    stNO_LENS[0].fEnergy := 5069.272832; stNO_LENS[0].fLow := 154.471527; stNO_LENS[0].fHigh := 156.009850; 
    stNO_LENS[1].fEnergy := 5079.421523; stNO_LENS[1].fLow := 153.906286; stNO_LENS[1].fHigh := 156.009850; 
    stNO_LENS[2].fEnergy := 5089.590532; stNO_LENS[2].fLow := 153.342381; stNO_LENS[2].fHigh := 156.009850; 
    stNO_LENS[3].fEnergy := 5099.779899; stNO_LENS[3].fLow := 152.779815; stNO_LENS[3].fHigh := 156.009850; 
    stNO_LENS[4].fEnergy := 5109.989665; stNO_LENS[4].fLow := 152.218592; stNO_LENS[4].fHigh := 156.009850; 
    stNO_LENS[5].fEnergy := 5120.219871; stNO_LENS[5].fLow := 151.658718; stNO_LENS[5].fHigh := 156.009850; 
    stNO_LENS[6].fEnergy := 5130.470558; stNO_LENS[6].fLow := 151.100196; stNO_LENS[6].fHigh := 156.009850; 
    stNO_LENS[7].fEnergy := 5140.741767; stNO_LENS[7].fLow := 150.543029; stNO_LENS[7].fHigh := 156.009850; 
    stNO_LENS[8].fEnergy := 5151.033539; stNO_LENS[8].fLow := 149.987222; stNO_LENS[8].fHigh := 156.009850; 
    stNO_LENS[9].fEnergy := 5161.345915; stNO_LENS[9].fLow := 149.432777; stNO_LENS[9].fHigh := 156.009850; 
    stNO_LENS[10].fEnergy := 5171.678936; stNO_LENS[10].fLow := 148.879700; stNO_LENS[10].fHigh := 156.009850; 
    stNO_LENS[11].fEnergy := 5182.032644; stNO_LENS[11].fLow := 148.327994; stNO_LENS[11].fHigh := 156.009850; 
    stNO_LENS[12].fEnergy := 5192.407080; stNO_LENS[12].fLow := 147.777661; stNO_LENS[12].fHigh := 156.009850; 
    stNO_LENS[13].fEnergy := 5202.802286; stNO_LENS[13].fLow := 147.228705; stNO_LENS[13].fHigh := 156.009850; 
    stNO_LENS[14].fEnergy := 5213.218304; stNO_LENS[14].fLow := 146.681131; stNO_LENS[14].fHigh := 156.009850; 
    stNO_LENS[15].fEnergy := 5223.655174; stNO_LENS[15].fLow := 146.134940; stNO_LENS[15].fHigh := 156.009850; 
    stNO_LENS[16].fEnergy := 5234.112938; stNO_LENS[16].fLow := 145.590136; stNO_LENS[16].fHigh := 156.022129; 
    stNO_LENS[17].fEnergy := 5244.591639; stNO_LENS[17].fLow := 145.046723; stNO_LENS[17].fHigh := 156.023236; 
    stNO_LENS[18].fEnergy := 5255.091319; stNO_LENS[18].fLow := 144.504703; stNO_LENS[18].fHigh := 156.013558; 
    stNO_LENS[19].fEnergy := 5265.612019; stNO_LENS[19].fLow := 143.964079; stNO_LENS[19].fHigh := 155.993480; 
    stNO_LENS[20].fEnergy := 5276.153781; stNO_LENS[20].fLow := 143.424854; stNO_LENS[20].fHigh := 155.963384; 
    stNO_LENS[21].fEnergy := 5286.716648; stNO_LENS[21].fLow := 142.887032; stNO_LENS[21].fHigh := 155.923643; 
    stNO_LENS[22].fEnergy := 5297.300661; stNO_LENS[22].fLow := 142.350614; stNO_LENS[22].fHigh := 155.874628; 
    stNO_LENS[23].fEnergy := 5307.905864; stNO_LENS[23].fLow := 141.815603; stNO_LENS[23].fHigh := 155.816705; 
    stNO_LENS[24].fEnergy := 5318.532299; stNO_LENS[24].fLow := 141.282002; stNO_LENS[24].fHigh := 155.750234; 
    stNO_LENS[25].fEnergy := 5329.180008; stNO_LENS[25].fLow := 140.749814; stNO_LENS[25].fHigh := 155.675570; 
    stNO_LENS[26].fEnergy := 5339.849033; stNO_LENS[26].fLow := 140.219040; stNO_LENS[26].fHigh := 155.593061; 
    stNO_LENS[27].fEnergy := 5350.539418; stNO_LENS[27].fLow := 139.689684; stNO_LENS[27].fHigh := 155.503052; 
    stNO_LENS[28].fEnergy := 5361.251205; stNO_LENS[28].fLow := 139.161747; stNO_LENS[28].fHigh := 155.405880; 
    stNO_LENS[29].fEnergy := 5371.984437; stNO_LENS[29].fLow := 138.635232; stNO_LENS[29].fHigh := 155.301878; 
    stNO_LENS[30].fEnergy := 5382.739157; stNO_LENS[30].fLow := 138.110142; stNO_LENS[30].fHigh := 155.191371; 
    stNO_LENS[31].fEnergy := 5393.515408; stNO_LENS[31].fLow := 137.586477; stNO_LENS[31].fHigh := 155.074681; 
    stNO_LENS[32].fEnergy := 5404.313233; stNO_LENS[32].fLow := 137.064240; stNO_LENS[32].fHigh := 154.952120; 
    stNO_LENS[33].fEnergy := 5415.132676; stNO_LENS[33].fLow := 136.543434; stNO_LENS[33].fHigh := 154.823998; 
    stNO_LENS[34].fEnergy := 5425.973779; stNO_LENS[34].fLow := 136.024059; stNO_LENS[34].fHigh := 154.690616; 
    stNO_LENS[35].fEnergy := 5436.836585; stNO_LENS[35].fLow := 135.506118; stNO_LENS[35].fHigh := 154.552270; 
    stNO_LENS[36].fEnergy := 5447.721139; stNO_LENS[36].fLow := 134.989613; stNO_LENS[36].fHigh := 154.409250; 
    stNO_LENS[37].fEnergy := 5458.627484; stNO_LENS[37].fLow := 134.474545; stNO_LENS[37].fHigh := 154.261839; 
    stNO_LENS[38].fEnergy := 5469.555664; stNO_LENS[38].fLow := 133.960916; stNO_LENS[38].fHigh := 154.110313; 
    stNO_LENS[39].fEnergy := 5480.505722; stNO_LENS[39].fLow := 133.448727; stNO_LENS[39].fHigh := 153.954945; 
    stNO_LENS[40].fEnergy := 5491.477701; stNO_LENS[40].fLow := 132.937980; stNO_LENS[40].fHigh := 153.795998; 
    stNO_LENS[41].fEnergy := 5502.471647; stNO_LENS[41].fLow := 132.428677; stNO_LENS[41].fHigh := 153.633731; 
    stNO_LENS[42].fEnergy := 5513.487603; stNO_LENS[42].fLow := 131.920818; stNO_LENS[42].fHigh := 153.468397; 
    stNO_LENS[43].fEnergy := 5524.525612; stNO_LENS[43].fLow := 131.414406; stNO_LENS[43].fHigh := 153.300240; 
    stNO_LENS[44].fEnergy := 5535.585720; stNO_LENS[44].fLow := 130.909441; stNO_LENS[44].fHigh := 153.129502; 
    stNO_LENS[45].fEnergy := 5546.667970; stNO_LENS[45].fLow := 130.405924; stNO_LENS[45].fHigh := 152.956416; 
    stNO_LENS[46].fEnergy := 5557.772406; stNO_LENS[46].fLow := 129.903857; stNO_LENS[46].fHigh := 152.781209; 
    stNO_LENS[47].fEnergy := 5568.899074; stNO_LENS[47].fLow := 129.403241; stNO_LENS[47].fHigh := 152.604103; 
    stNO_LENS[48].fEnergy := 5580.048018; stNO_LENS[48].fLow := 128.904077; stNO_LENS[48].fHigh := 152.425314; 
    stNO_LENS[49].fEnergy := 5591.219281; stNO_LENS[49].fLow := 128.406365; stNO_LENS[49].fHigh := 152.245051; 
    stNO_LENS[50].fEnergy := 5602.412910; stNO_LENS[50].fLow := 127.910107; stNO_LENS[50].fHigh := 152.063517; 
    stNO_LENS[51].fEnergy := 5613.628948; stNO_LENS[51].fLow := 127.415303; stNO_LENS[51].fHigh := 151.880912; 
    stNO_LENS[52].fEnergy := 5624.867440; stNO_LENS[52].fLow := 126.921955; stNO_LENS[52].fHigh := 151.697425; 
    stNO_LENS[53].fEnergy := 5636.128433; stNO_LENS[53].fLow := 126.430063; stNO_LENS[53].fHigh := 151.513245; 
    stNO_LENS[54].fEnergy := 5647.411969; stNO_LENS[54].fLow := 125.939627; stNO_LENS[54].fHigh := 151.328551; 
    stNO_LENS[55].fEnergy := 5658.718095; stNO_LENS[55].fLow := 125.450648; stNO_LENS[55].fHigh := 151.143518; 
    stNO_LENS[56].fEnergy := 5670.046857; stNO_LENS[56].fLow := 124.963127; stNO_LENS[56].fHigh := 150.958316; 
    stNO_LENS[57].fEnergy := 5681.398298; stNO_LENS[57].fLow := 124.477064; stNO_LENS[57].fHigh := 150.773109; 
    stNO_LENS[58].fEnergy := 5692.772465; stNO_LENS[58].fLow := 123.992460; stNO_LENS[58].fHigh := 150.588055; 
    stNO_LENS[59].fEnergy := 5704.169403; stNO_LENS[59].fLow := 123.509315; stNO_LENS[59].fHigh := 150.403307; 
    stNO_LENS[60].fEnergy := 5715.589158; stNO_LENS[60].fLow := 123.027630; stNO_LENS[60].fHigh := 150.219012; 
    stNO_LENS[61].fEnergy := 5727.031775; stNO_LENS[61].fLow := 122.547404; stNO_LENS[61].fHigh := 150.035315; 
    stNO_LENS[62].fEnergy := 5738.497300; stNO_LENS[62].fLow := 122.068638; stNO_LENS[62].fHigh := 149.852352; 
    stNO_LENS[63].fEnergy := 5749.985779; stNO_LENS[63].fLow := 121.591332; stNO_LENS[63].fHigh := 149.670256; 
    stNO_LENS[64].fEnergy := 5761.497259; stNO_LENS[64].fLow := 121.115486; stNO_LENS[64].fHigh := 149.489154; 
    stNO_LENS[65].fEnergy := 5773.031784; stNO_LENS[65].fLow := 120.641101; stNO_LENS[65].fHigh := 149.309169; 
    stNO_LENS[66].fEnergy := 5784.589401; stNO_LENS[66].fLow := 120.168176; stNO_LENS[66].fHigh := 149.130419; 
    stNO_LENS[67].fEnergy := 5796.170157; stNO_LENS[67].fLow := 119.696711; stNO_LENS[67].fHigh := 148.953017; 
    stNO_LENS[68].fEnergy := 5807.774097; stNO_LENS[68].fLow := 119.226706; stNO_LENS[68].fHigh := 148.777072; 
    stNO_LENS[69].fEnergy := 5819.401269; stNO_LENS[69].fLow := 118.758161; stNO_LENS[69].fHigh := 148.602686; 
    stNO_LENS[70].fEnergy := 5831.051718; stNO_LENS[70].fLow := 118.291076; stNO_LENS[70].fHigh := 148.429960; 
    stNO_LENS[71].fEnergy := 5842.725491; stNO_LENS[71].fLow := 117.825451; stNO_LENS[71].fHigh := 148.258988; 
    stNO_LENS[72].fEnergy := 5854.422635; stNO_LENS[72].fLow := 117.361285; stNO_LENS[72].fHigh := 148.089861; 
    stNO_LENS[73].fEnergy := 5866.143197; stNO_LENS[73].fLow := 116.898578; stNO_LENS[73].fHigh := 147.922666; 
    stNO_LENS[74].fEnergy := 5877.887224; stNO_LENS[74].fLow := 116.437330; stNO_LENS[74].fHigh := 147.757483; 
    stNO_LENS[75].fEnergy := 5889.654762; stNO_LENS[75].fLow := 115.977540; stNO_LENS[75].fHigh := 147.594392; 
    stNO_LENS[76].fEnergy := 5901.445859; stNO_LENS[76].fLow := 115.519207; stNO_LENS[76].fHigh := 147.433465; 
    stNO_LENS[77].fEnergy := 5913.260561; stNO_LENS[77].fLow := 115.062332; stNO_LENS[77].fHigh := 147.274774; 
    stNO_LENS[78].fEnergy := 5925.098917; stNO_LENS[78].fLow := 114.606914; stNO_LENS[78].fHigh := 147.118383; 
    stNO_LENS[79].fEnergy := 5936.960973; stNO_LENS[79].fLow := 114.152952; stNO_LENS[79].fHigh := 146.964356; 
    stNO_LENS[80].fEnergy := 5948.846776; stNO_LENS[80].fLow := 113.700445; stNO_LENS[80].fHigh := 146.812749; 
    stNO_LENS[81].fEnergy := 5960.756375; stNO_LENS[81].fLow := 113.249392; stNO_LENS[81].fHigh := 146.663619; 
    stNO_LENS[82].fEnergy := 5972.689818; stNO_LENS[82].fLow := 112.799794; stNO_LENS[82].fHigh := 146.517015; 
    stNO_LENS[83].fEnergy := 5984.647151; stNO_LENS[83].fLow := 112.351649; stNO_LENS[83].fHigh := 146.372987; 
    stNO_LENS[84].fEnergy := 5996.628422; stNO_LENS[84].fLow := 111.904956; stNO_LENS[84].fHigh := 146.231576; 
    stNO_LENS[85].fEnergy := 6008.633680; stNO_LENS[85].fLow := 111.459715; stNO_LENS[85].fHigh := 146.092825; 
    stNO_LENS[86].fEnergy := 6020.662973; stNO_LENS[86].fLow := 111.015925; stNO_LENS[86].fHigh := 145.956770; 
    stNO_LENS[87].fEnergy := 6032.716348; stNO_LENS[87].fLow := 110.573584; stNO_LENS[87].fHigh := 145.823445; 
    stNO_LENS[88].fEnergy := 6044.793854; stNO_LENS[88].fLow := 110.132692; stNO_LENS[88].fHigh := 145.692881; 
    stNO_LENS[89].fEnergy := 6056.895540; stNO_LENS[89].fLow := 109.693247; stNO_LENS[89].fHigh := 145.565105; 
    stNO_LENS[90].fEnergy := 6069.021453; stNO_LENS[90].fLow := 109.255249; stNO_LENS[90].fHigh := 145.440142; 
    stNO_LENS[91].fEnergy := 6081.171642; stNO_LENS[91].fLow := 108.818697; stNO_LENS[91].fHigh := 145.318013; 
    stNO_LENS[92].fEnergy := 6093.346156; stNO_LENS[92].fLow := 108.383589; stNO_LENS[92].fHigh := 145.198736; 
    stNO_LENS[93].fEnergy := 6105.545043; stNO_LENS[93].fLow := 107.949924; stNO_LENS[93].fHigh := 145.082327; 
    stNO_LENS[94].fEnergy := 6117.768352; stNO_LENS[94].fLow := 107.517701; stNO_LENS[94].fHigh := 144.968799; 
    stNO_LENS[95].fEnergy := 6130.016132; stNO_LENS[95].fLow := 107.086918; stNO_LENS[95].fHigh := 144.858160; 
    stNO_LENS[96].fEnergy := 6142.288433; stNO_LENS[96].fLow := 106.657575; stNO_LENS[96].fHigh := 144.750419; 
    stNO_LENS[97].fEnergy := 6154.585303; stNO_LENS[97].fLow := 106.229670; stNO_LENS[97].fHigh := 144.645579; 
    stNO_LENS[98].fEnergy := 6166.906791; stNO_LENS[98].fLow := 105.803201; stNO_LENS[98].fHigh := 144.543642; 
    stNO_LENS[99].fEnergy := 6179.252946; stNO_LENS[99].fLow := 105.378168; stNO_LENS[99].fHigh := 144.444606; 
    stNO_LENS[100].fEnergy := 6191.623819; stNO_LENS[100].fLow := 104.954569; stNO_LENS[100].fHigh := 144.348469; 
    stNO_LENS[101].fEnergy := 6204.019458; stNO_LENS[101].fLow := 104.532401; stNO_LENS[101].fHigh := 144.255225; 
    stNO_LENS[102].fEnergy := 6216.439913; stNO_LENS[102].fLow := 104.111665; stNO_LENS[102].fHigh := 144.164864; 
    stNO_LENS[103].fEnergy := 6228.885234; stNO_LENS[103].fLow := 103.692358; stNO_LENS[103].fHigh := 144.077376; 
    stNO_LENS[104].fEnergy := 6241.355471; stNO_LENS[104].fLow := 103.274478; stNO_LENS[104].fHigh := 143.992747; 
    stNO_LENS[105].fEnergy := 6253.850673; stNO_LENS[105].fLow := 102.858024; stNO_LENS[105].fHigh := 143.910962; 
    stNO_LENS[106].fEnergy := 6266.370890; stNO_LENS[106].fLow := 102.442995; stNO_LENS[106].fHigh := 143.832003; 
    stNO_LENS[107].fEnergy := 6278.916173; stNO_LENS[107].fLow := 102.029389; stNO_LENS[107].fHigh := 143.755850; 
    stNO_LENS[108].fEnergy := 6291.486572; stNO_LENS[108].fLow := 101.617203; stNO_LENS[108].fHigh := 143.682481; 
    stNO_LENS[109].fEnergy := 6304.082136; stNO_LENS[109].fLow := 101.206436; stNO_LENS[109].fHigh := 143.611870; 
    stNO_LENS[110].fEnergy := 6316.702917; stNO_LENS[110].fLow := 100.797087; stNO_LENS[110].fHigh := 143.543993; 
    stNO_LENS[111].fEnergy := 6329.348965; stNO_LENS[111].fLow := 100.389154; stNO_LENS[111].fHigh := 143.478819; 
    stNO_LENS[112].fEnergy := 6342.020330; stNO_LENS[112].fLow := 99.982634; stNO_LENS[112].fHigh := 143.416319; 
    stNO_LENS[113].fEnergy := 6354.717063; stNO_LENS[113].fLow := 99.577526; stNO_LENS[113].fHigh := 143.356460; 
    stNO_LENS[114].fEnergy := 6367.439215; stNO_LENS[114].fLow := 99.173828; stNO_LENS[114].fHigh := 143.299207; 
    stNO_LENS[115].fEnergy := 6380.186837; stNO_LENS[115].fLow := 98.771538; stNO_LENS[115].fHigh := 143.244524; 
    stNO_LENS[116].fEnergy := 6392.959979; stNO_LENS[116].fLow := 98.370654; stNO_LENS[116].fHigh := 143.192372; 
    stNO_LENS[117].fEnergy := 6405.758694; stNO_LENS[117].fLow := 97.971174; stNO_LENS[117].fHigh := 143.142713; 
    stNO_LENS[118].fEnergy := 6418.583031; stNO_LENS[118].fLow := 97.573096; stNO_LENS[118].fHigh := 143.095503; 
    stNO_LENS[119].fEnergy := 6431.433043; stNO_LENS[119].fLow := 97.176418; stNO_LENS[119].fHigh := 143.050699; 
    stNO_LENS[120].fEnergy := 6444.308780; stNO_LENS[120].fLow := 96.781138; stNO_LENS[120].fHigh := 143.008256; 
    stNO_LENS[121].fEnergy := 6457.210295; stNO_LENS[121].fLow := 96.387254; stNO_LENS[121].fHigh := 142.968127; 
    stNO_LENS[122].fEnergy := 6470.137639; stNO_LENS[122].fLow := 95.994763; stNO_LENS[122].fHigh := 142.930263; 
    stNO_LENS[123].fEnergy := 6483.090863; stNO_LENS[123].fLow := 95.603664; stNO_LENS[123].fHigh := 142.894614; 
    stNO_LENS[124].fEnergy := 6496.070019; stNO_LENS[124].fLow := 95.213954; stNO_LENS[124].fHigh := 142.861129; 
    stNO_LENS[125].fEnergy := 6509.075160; stNO_LENS[125].fLow := 94.825631; stNO_LENS[125].fHigh := 142.829753; 
    stNO_LENS[126].fEnergy := 6522.106337; stNO_LENS[126].fLow := 94.438693; stNO_LENS[126].fHigh := 142.800431; 
    stNO_LENS[127].fEnergy := 6535.163603; stNO_LENS[127].fLow := 94.053137; stNO_LENS[127].fHigh := 142.773109; 
    stNO_LENS[128].fEnergy := 6548.247009; stNO_LENS[128].fLow := 93.668962; stNO_LENS[128].fHigh := 142.747727; 
    stNO_LENS[129].fEnergy := 6561.356609; stNO_LENS[129].fLow := 93.286164; stNO_LENS[129].fHigh := 142.724228; 
    stNO_LENS[130].fEnergy := 6574.492453; stNO_LENS[130].fLow := 92.904742; stNO_LENS[130].fHigh := 142.702549; 
    stNO_LENS[131].fEnergy := 6587.654596; stNO_LENS[131].fLow := 92.524694; stNO_LENS[131].fHigh := 142.682630; 
    stNO_LENS[132].fEnergy := 6600.843089; stNO_LENS[132].fLow := 92.146016; stNO_LENS[132].fHigh := 142.664407; 
    stNO_LENS[133].fEnergy := 6614.057986; stNO_LENS[133].fLow := 91.768706; stNO_LENS[133].fHigh := 142.647816; 
    stNO_LENS[134].fEnergy := 6627.299339; stNO_LENS[134].fLow := 91.392763; stNO_LENS[134].fHigh := 142.632791; 
    stNO_LENS[135].fEnergy := 6640.567201; stNO_LENS[135].fLow := 91.018183; stNO_LENS[135].fHigh := 142.619266; 
    stNO_LENS[136].fEnergy := 6653.861625; stNO_LENS[136].fLow := 90.644964; stNO_LENS[136].fHigh := 142.607171; 
    stNO_LENS[137].fEnergy := 6667.182665; stNO_LENS[137].fLow := 90.273103; stNO_LENS[137].fHigh := 142.596440; 
    stNO_LENS[138].fEnergy := 6680.530374; stNO_LENS[138].fLow := 89.902598; stNO_LENS[138].fHigh := 142.587000; 
    stNO_LENS[139].fEnergy := 6693.904804; stNO_LENS[139].fLow := 89.533447; stNO_LENS[139].fHigh := 142.578781; 
    stNO_LENS[140].fEnergy := 6707.306011; stNO_LENS[140].fLow := 89.165646; stNO_LENS[140].fHigh := 142.571711; 
    stNO_LENS[141].fEnergy := 6720.734046; stNO_LENS[141].fLow := 88.799194; stNO_LENS[141].fHigh := 142.565716; 
    stNO_LENS[142].fEnergy := 6734.188965; stNO_LENS[142].fLow := 88.434088; stNO_LENS[142].fHigh := 142.560721; 
    stNO_LENS[143].fEnergy := 6747.670820; stNO_LENS[143].fLow := 88.070324; stNO_LENS[143].fHigh := 142.556653; 
    stNO_LENS[144].fEnergy := 6761.179666; stNO_LENS[144].fLow := 87.707901; stNO_LENS[144].fHigh := 142.553434; 
    stNO_LENS[145].fEnergy := 6774.715557; stNO_LENS[145].fLow := 87.346815; stNO_LENS[145].fHigh := 142.550988; 
    stNO_LENS[146].fEnergy := 6788.278546; stNO_LENS[146].fLow := 86.987064; stNO_LENS[146].fHigh := 142.549237; 
    stNO_LENS[147].fEnergy := 6801.868689; stNO_LENS[147].fLow := 86.628646; stNO_LENS[147].fHigh := 142.548102; 
    stNO_LENS[148].fEnergy := 6815.486039; stNO_LENS[148].fLow := 86.271557; stNO_LENS[148].fHigh := 142.547505; 
    stNO_LENS[149].fEnergy := 6829.130652; stNO_LENS[149].fLow := 85.915795; stNO_LENS[149].fHigh := 142.547365; 
    stNO_LENS[150].fEnergy := 6842.802580; stNO_LENS[150].fLow := 85.561357; stNO_LENS[150].fHigh := 142.547602; 
    stNO_LENS[151].fEnergy := 6856.501880; stNO_LENS[151].fLow := 85.208240; stNO_LENS[151].fHigh := 142.548134; 
    stNO_LENS[152].fEnergy := 6870.228606; stNO_LENS[152].fLow := 84.856441; stNO_LENS[152].fHigh := 142.548880; 
    stNO_LENS[153].fEnergy := 6883.982813; stNO_LENS[153].fLow := 84.505959; stNO_LENS[153].fHigh := 142.549757; 
    stNO_LENS[154].fEnergy := 6897.764556; stNO_LENS[154].fLow := 84.156788; stNO_LENS[154].fHigh := 142.550682; 
    stNO_LENS[155].fEnergy := 6911.573889; stNO_LENS[155].fLow := 83.808928; stNO_LENS[155].fHigh := 142.551572; 
    stNO_LENS[156].fEnergy := 6925.410870; stNO_LENS[156].fLow := 83.462375; stNO_LENS[156].fHigh := 142.552342; 
    stNO_LENS[157].fEnergy := 6939.275551; stNO_LENS[157].fLow := 83.117126; stNO_LENS[157].fHigh := 142.552910; 
    stNO_LENS[158].fEnergy := 6953.167990; stNO_LENS[158].fLow := 82.773178; stNO_LENS[158].fHigh := 142.553189; 
    stNO_LENS[159].fEnergy := 6967.088242; stNO_LENS[159].fLow := 82.430528; stNO_LENS[159].fHigh := 142.553096; 
    stNO_LENS[160].fEnergy := 6981.036362; stNO_LENS[160].fLow := 82.089174; stNO_LENS[160].fHigh := 142.552545; 
    stNO_LENS[161].fEnergy := 6995.012406; stNO_LENS[161].fLow := 81.749112; stNO_LENS[161].fHigh := 142.551451; 
    stNO_LENS[162].fEnergy := 7009.016430; stNO_LENS[162].fLow := 81.410340; stNO_LENS[162].fHigh := 142.549728; 
    stNO_LENS[163].fEnergy := 7023.048490; stNO_LENS[163].fLow := 81.072854; stNO_LENS[163].fHigh := 142.547290; 
    stNO_LENS[164].fEnergy := 7037.108643; stNO_LENS[164].fLow := 80.736651; stNO_LENS[164].fHigh := 142.544051; 
    stNO_LENS[165].fEnergy := 7051.196944; stNO_LENS[165].fLow := 80.401730; stNO_LENS[165].fHigh := 142.539926; 
    stNO_LENS[166].fEnergy := 7065.313449; stNO_LENS[166].fLow := 80.068085; stNO_LENS[166].fHigh := 142.534829; 
    stNO_LENS[167].fEnergy := 7079.458216; stNO_LENS[167].fLow := 79.735715; stNO_LENS[167].fHigh := 142.528674; 
    stNO_LENS[168].fEnergy := 7093.631301; stNO_LENS[168].fLow := 79.404617; stNO_LENS[168].fHigh := 142.521375; 
    stNO_LENS[169].fEnergy := 7107.832760; stNO_LENS[169].fLow := 79.074786; stNO_LENS[169].fHigh := 142.512847; 
    stNO_LENS[170].fEnergy := 7122.062651; stNO_LENS[170].fLow := 78.746221; stNO_LENS[170].fHigh := 142.503004; 
    stNO_LENS[171].fEnergy := 7136.321030; stNO_LENS[171].fLow := 78.418918; stNO_LENS[171].fHigh := 142.491760; 
    stNO_LENS[172].fEnergy := 7150.607954; stNO_LENS[172].fLow := 78.092875; stNO_LENS[172].fHigh := 142.479032; 
    stNO_LENS[173].fEnergy := 7164.923481; stNO_LENS[173].fLow := 77.768087; stNO_LENS[173].fHigh := 142.464734; 
    stNO_LENS[174].fEnergy := 7179.267667; stNO_LENS[174].fLow := 77.444552; stNO_LENS[174].fHigh := 142.448782; 
    stNO_LENS[175].fEnergy := 7193.640571; stNO_LENS[175].fLow := 77.122267; stNO_LENS[175].fHigh := 142.431092; 
    stNO_LENS[176].fEnergy := 7208.042249; stNO_LENS[176].fLow := 76.801228; stNO_LENS[176].fHigh := 142.411581; 
    stNO_LENS[177].fEnergy := 7222.472759; stNO_LENS[177].fLow := 76.481433; stNO_LENS[177].fHigh := 142.390166; 
    stNO_LENS[178].fEnergy := 7236.932159; stNO_LENS[178].fLow := 76.162878; stNO_LENS[178].fHigh := 142.366765; 
    stNO_LENS[179].fEnergy := 7251.420507; stNO_LENS[179].fLow := 75.845560; stNO_LENS[179].fHigh := 142.341297; 
    stNO_LENS[180].fEnergy := 7265.937860; stNO_LENS[180].fLow := 75.529476; stNO_LENS[180].fHigh := 142.313679; 
    stNO_LENS[181].fEnergy := 7280.484278; stNO_LENS[181].fLow := 75.214623; stNO_LENS[181].fHigh := 142.283833; 
    stNO_LENS[182].fEnergy := 7295.059817; stNO_LENS[182].fLow := 74.900997; stNO_LENS[182].fHigh := 142.251678; 
    stNO_LENS[183].fEnergy := 7309.664536; stNO_LENS[183].fLow := 74.588595; stNO_LENS[183].fHigh := 142.217136; 
    stNO_LENS[184].fEnergy := 7324.298495; stNO_LENS[184].fLow := 74.277415; stNO_LENS[184].fHigh := 142.180129; 
    stNO_LENS[185].fEnergy := 7338.961750; stNO_LENS[185].fLow := 73.967452; stNO_LENS[185].fHigh := 142.140581; 
    stNO_LENS[186].fEnergy := 7353.654361; stNO_LENS[186].fLow := 73.658704; stNO_LENS[186].fHigh := 142.098415; 
    stNO_LENS[187].fEnergy := 7368.376387; stNO_LENS[187].fLow := 73.351168; stNO_LENS[187].fHigh := 142.053558; 
    stNO_LENS[188].fEnergy := 7383.127886; stNO_LENS[188].fLow := 73.044839; stNO_LENS[188].fHigh := 142.005934; 
    stNO_LENS[189].fEnergy := 7397.908918; stNO_LENS[189].fLow := 72.739716; stNO_LENS[189].fHigh := 141.955472; 
    stNO_LENS[190].fEnergy := 7412.719542; stNO_LENS[190].fLow := 72.435793; stNO_LENS[190].fHigh := 141.902101; 
    stNO_LENS[191].fEnergy := 7427.559816; stNO_LENS[191].fLow := 72.133070; stNO_LENS[191].fHigh := 141.845750; 
    stNO_LENS[192].fEnergy := 7442.429801; stNO_LENS[192].fLow := 71.831541; stNO_LENS[192].fHigh := 141.786350; 
    stNO_LENS[193].fEnergy := 7457.329555; stNO_LENS[193].fLow := 71.531203; stNO_LENS[193].fHigh := 141.723834; 
    stNO_LENS[194].fEnergy := 7472.259139; stNO_LENS[194].fLow := 71.232055; stNO_LENS[194].fHigh := 141.658137; 
    stNO_LENS[195].fEnergy := 7487.218612; stNO_LENS[195].fLow := 70.934091; stNO_LENS[195].fHigh := 141.589194; 
    stNO_LENS[196].fEnergy := 7502.208033; stNO_LENS[196].fLow := 70.637309; stNO_LENS[196].fHigh := 141.516941; 
    stNO_LENS[197].fEnergy := 7517.227464; stNO_LENS[197].fLow := 70.341705; stNO_LENS[197].fHigh := 141.441317; 
    stNO_LENS[198].fEnergy := 7532.276963; stNO_LENS[198].fLow := 70.047277; stNO_LENS[198].fHigh := 141.362263; 
    stNO_LENS[199].fEnergy := 7547.356592; stNO_LENS[199].fLow := 69.754020; stNO_LENS[199].fHigh := 141.279720; 
    stNO_LENS[200].fEnergy := 7562.466410; stNO_LENS[200].fLow := 69.461932; stNO_LENS[200].fHigh := 141.193632; 
    stNO_LENS[201].fEnergy := 7577.606478; stNO_LENS[201].fLow := 69.171009; stNO_LENS[201].fHigh := 141.103944; 
    stNO_LENS[202].fEnergy := 7592.776856; stNO_LENS[202].fLow := 68.881248; stNO_LENS[202].fHigh := 141.010603; 
    stNO_LENS[203].fEnergy := 7607.977605; stNO_LENS[203].fLow := 68.592645; stNO_LENS[203].fHigh := 140.913560; 
    stNO_LENS[204].fEnergy := 7623.208787; stNO_LENS[204].fLow := 68.305197; stNO_LENS[204].fHigh := 140.812763; 
    stNO_LENS[205].fEnergy := 7638.470461; stNO_LENS[205].fLow := 68.018901; stNO_LENS[205].fHigh := 140.708168; 
    stNO_LENS[206].fEnergy := 7653.762689; stNO_LENS[206].fLow := 67.733753; stNO_LENS[206].fHigh := 140.599727; 
    stNO_LENS[207].fEnergy := 7669.085532; stNO_LENS[207].fLow := 67.449750; stNO_LENS[207].fHigh := 140.487400; 
    stNO_LENS[208].fEnergy := 7684.439051; stNO_LENS[208].fLow := 67.166889; stNO_LENS[208].fHigh := 140.371143; 
    stNO_LENS[209].fEnergy := 7699.823309; stNO_LENS[209].fLow := 66.885165; stNO_LENS[209].fHigh := 140.250920; 
    stNO_LENS[210].fEnergy := 7715.238365; stNO_LENS[210].fLow := 66.604577; stNO_LENS[210].fHigh := 140.126694; 
    stNO_LENS[211].fEnergy := 7730.684283; stNO_LENS[211].fLow := 66.325120; stNO_LENS[211].fHigh := 139.998430; 
    stNO_LENS[212].fEnergy := 7746.161123; stNO_LENS[212].fLow := 66.046791; stNO_LENS[212].fHigh := 139.866096; 
    stNO_LENS[213].fEnergy := 7761.668948; stNO_LENS[213].fLow := 65.769586; stNO_LENS[213].fHigh := 139.729663; 
    stNO_LENS[214].fEnergy := 7777.207819; stNO_LENS[214].fLow := 65.493503; stNO_LENS[214].fHigh := 139.589104; 
    stNO_LENS[215].fEnergy := 7792.777800; stNO_LENS[215].fLow := 65.218537; stNO_LENS[215].fHigh := 139.444394; 
    stNO_LENS[216].fEnergy := 7808.378951; stNO_LENS[216].fLow := 64.944686; stNO_LENS[216].fHigh := 139.295510; 
    stNO_LENS[217].fEnergy := 7824.011336; stNO_LENS[217].fLow := 64.671946; stNO_LENS[217].fHigh := 139.142433; 
    stNO_LENS[218].fEnergy := 7839.675018; stNO_LENS[218].fLow := 64.400313; stNO_LENS[218].fHigh := 138.985145; 
    stNO_LENS[219].fEnergy := 7855.370057; stNO_LENS[219].fLow := 64.129785; stNO_LENS[219].fHigh := 138.823631; 
    stNO_LENS[220].fEnergy := 7871.096519; stNO_LENS[220].fLow := 63.860357; stNO_LENS[220].fHigh := 138.657880; 
    stNO_LENS[221].fEnergy := 7886.854464; stNO_LENS[221].fLow := 63.592027; stNO_LENS[221].fHigh := 138.487882; 
    stNO_LENS[222].fEnergy := 7902.643958; stNO_LENS[222].fLow := 63.324790; stNO_LENS[222].fHigh := 138.313630; 
    stNO_LENS[223].fEnergy := 7918.465061; stNO_LENS[223].fLow := 63.058644; stNO_LENS[223].fHigh := 138.135119; 
    stNO_LENS[224].fEnergy := 7934.317839; stNO_LENS[224].fLow := 62.793585; stNO_LENS[224].fHigh := 137.952349; 
    stNO_LENS[225].fEnergy := 7950.202354; stNO_LENS[225].fLow := 62.529610; stNO_LENS[225].fHigh := 137.765320; 
    stNO_LENS[226].fEnergy := 7966.118670; stNO_LENS[226].fLow := 62.266715; stNO_LENS[226].fHigh := 137.608060; 
    stNO_LENS[227].fEnergy := 7982.066850; stNO_LENS[227].fLow := 62.004896; stNO_LENS[227].fHigh := 137.048845; 
    stNO_LENS[228].fEnergy := 7998.046958; stNO_LENS[228].fLow := 61.744151; stNO_LENS[228].fHigh := 136.491790; 
    stNO_LENS[229].fEnergy := 8014.059059; stNO_LENS[229].fLow := 61.484476; stNO_LENS[229].fHigh := 135.936902; 
    stNO_LENS[230].fEnergy := 8030.103216; stNO_LENS[230].fLow := 61.225868; stNO_LENS[230].fHigh := 135.384186; 
    stNO_LENS[231].fEnergy := 8046.179493; stNO_LENS[231].fLow := 60.968322; stNO_LENS[231].fHigh := 134.833648; 
    stNO_LENS[232].fEnergy := 8062.287955; stNO_LENS[232].fLow := 60.711836; stNO_LENS[232].fHigh := 134.285293; 
    stNO_LENS[233].fEnergy := 8078.428667; stNO_LENS[233].fLow := 60.456407; stNO_LENS[233].fHigh := 133.739125; 
    stNO_LENS[234].fEnergy := 8094.601692; stNO_LENS[234].fLow := 60.202030; stNO_LENS[234].fHigh := 133.195147; 
    stNO_LENS[235].fEnergy := 8110.807095; stNO_LENS[235].fLow := 59.948702; stNO_LENS[235].fHigh := 132.653363; 
    stNO_LENS[236].fEnergy := 8127.044942; stNO_LENS[236].fLow := 59.696420; stNO_LENS[236].fHigh := 132.113775; 
    stNO_LENS[237].fEnergy := 8143.315296; stNO_LENS[237].fLow := 59.445181; stNO_LENS[237].fHigh := 131.576385; 
    stNO_LENS[238].fEnergy := 8159.618224; stNO_LENS[238].fLow := 59.194981; stNO_LENS[238].fHigh := 131.041195; 
    stNO_LENS[239].fEnergy := 8175.953791; stNO_LENS[239].fLow := 58.945817; stNO_LENS[239].fHigh := 130.508206; 
    stNO_LENS[240].fEnergy := 8192.322061; stNO_LENS[240].fLow := 58.697684; stNO_LENS[240].fHigh := 129.977418; 
    stNO_LENS[241].fEnergy := 8208.723101; stNO_LENS[241].fLow := 58.450581; stNO_LENS[241].fHigh := 129.448832; 
    stNO_LENS[242].fEnergy := 8225.156976; stNO_LENS[242].fLow := 58.204503; stNO_LENS[242].fHigh := 128.922447; 
    stNO_LENS[243].fEnergy := 8241.623751; stNO_LENS[243].fLow := 57.959446; stNO_LENS[243].fHigh := 128.398263; 
    stNO_LENS[244].fEnergy := 8258.123493; stNO_LENS[244].fLow := 57.715408; stNO_LENS[244].fHigh := 127.876278; 
    stNO_LENS[245].fEnergy := 8274.656267; stNO_LENS[245].fLow := 57.472386; stNO_LENS[245].fHigh := 127.356491; 
    stNO_LENS[246].fEnergy := 8291.222140; stNO_LENS[246].fLow := 57.230375; stNO_LENS[246].fHigh := 126.838900; 
    stNO_LENS[247].fEnergy := 8307.821178; stNO_LENS[247].fLow := 56.989372; stNO_LENS[247].fHigh := 126.323503; 
    stNO_LENS[248].fEnergy := 8324.453447; stNO_LENS[248].fLow := 56.749374; stNO_LENS[248].fHigh := 125.810298; 
    stNO_LENS[249].fEnergy := 8341.119014; stNO_LENS[249].fLow := 56.510377; stNO_LENS[249].fHigh := 125.299281; 
    stNO_LENS[250].fEnergy := 8357.817945; stNO_LENS[250].fLow := 56.272379; stNO_LENS[250].fHigh := 124.790450; 
    stNO_LENS[251].fEnergy := 8374.550308; stNO_LENS[251].fLow := 56.035375; stNO_LENS[251].fHigh := 124.283800; 
    stNO_LENS[252].fEnergy := 8391.316169; stNO_LENS[252].fLow := 55.799362; stNO_LENS[252].fHigh := 123.779328; 
    stNO_LENS[253].fEnergy := 8408.115595; stNO_LENS[253].fLow := 55.564337; stNO_LENS[253].fHigh := 123.277031; 
    stNO_LENS[254].fEnergy := 8424.948653; stNO_LENS[254].fLow := 55.330296; stNO_LENS[254].fHigh := 122.776902; 
    stNO_LENS[255].fEnergy := 8441.815412; stNO_LENS[255].fLow := 55.097236; stNO_LENS[255].fHigh := 122.278938; 
    stNO_LENS[256].fEnergy := 8458.715938; stNO_LENS[256].fLow := 54.865154; stNO_LENS[256].fHigh := 121.783134; 
    stNO_LENS[257].fEnergy := 8475.650298; stNO_LENS[257].fLow := 54.634046; stNO_LENS[257].fHigh := 121.289485; 
    stNO_LENS[258].fEnergy := 8492.618561; stNO_LENS[258].fLow := 54.403909; stNO_LENS[258].fHigh := 120.797985; 
    stNO_LENS[259].fEnergy := 8509.620795; stNO_LENS[259].fLow := 54.174739; stNO_LENS[259].fHigh := 120.308629; 
    stNO_LENS[260].fEnergy := 8526.657067; stNO_LENS[260].fLow := 53.946533; stNO_LENS[260].fHigh := 119.821410; 
    stNO_LENS[261].fEnergy := 8543.727446; stNO_LENS[261].fLow := 53.719288; stNO_LENS[261].fHigh := 119.336324; 
    stNO_LENS[262].fEnergy := 8560.832000; stNO_LENS[262].fLow := 53.493000; stNO_LENS[262].fHigh := 118.853363; 
    stNO_LENS[263].fEnergy := 8577.970797; stNO_LENS[263].fLow := 53.267666; stNO_LENS[263].fHigh := 118.372521; 
    stNO_LENS[264].fEnergy := 8595.143906; stNO_LENS[264].fLow := 53.043282; stNO_LENS[264].fHigh := 117.893792; 
    stNO_LENS[265].fEnergy := 8612.351395; stNO_LENS[265].fLow := 52.819845; stNO_LENS[265].fHigh := 117.417168; 
    stNO_LENS[266].fEnergy := 8629.593334; stNO_LENS[266].fLow := 52.597352; stNO_LENS[266].fHigh := 116.942644; 
    stNO_LENS[267].fEnergy := 8646.869792; stNO_LENS[267].fLow := 52.375800; stNO_LENS[267].fHigh := 116.470212; 
    stNO_LENS[268].fEnergy := 8664.180837; stNO_LENS[268].fLow := 52.155184; stNO_LENS[268].fHigh := 115.999864; 
    stNO_LENS[269].fEnergy := 8681.526538; stNO_LENS[269].fLow := 51.935503; stNO_LENS[269].fHigh := 115.531593; 
    stNO_LENS[270].fEnergy := 8698.906966; stNO_LENS[270].fLow := 51.716751; stNO_LENS[270].fHigh := 115.065393; 
    stNO_LENS[271].fEnergy := 8716.322189; stNO_LENS[271].fLow := 51.498926; stNO_LENS[271].fHigh := 114.601255; 
    stNO_LENS[272].fEnergy := 8733.772278; stNO_LENS[272].fLow := 51.282026; stNO_LENS[272].fHigh := 114.139171; 
    stNO_LENS[273].fEnergy := 8751.257302; stNO_LENS[273].fLow := 51.066045; stNO_LENS[273].fHigh := 113.679134; 
    stNO_LENS[274].fEnergy := 8768.777330; stNO_LENS[274].fLow := 50.850981; stNO_LENS[274].fHigh := 113.221136; 
    stNO_LENS[275].fEnergy := 8786.332434; stNO_LENS[275].fLow := 50.636831; stNO_LENS[275].fHigh := 112.765169; 
    stNO_LENS[276].fEnergy := 8803.922684; stNO_LENS[276].fLow := 50.423591; stNO_LENS[276].fHigh := 112.311224; 
    stNO_LENS[277].fEnergy := 8821.548149; stNO_LENS[277].fLow := 50.211258; stNO_LENS[277].fHigh := 111.859294; 
    stNO_LENS[278].fEnergy := 8839.208900; stNO_LENS[278].fLow := 49.999829; stNO_LENS[278].fHigh := 111.409371; 
    stNO_LENS[279].fEnergy := 8856.905008; stNO_LENS[279].fLow := 49.789301; stNO_LENS[279].fHigh := 110.961445; 
    stNO_LENS[280].fEnergy := 8874.636543; stNO_LENS[280].fLow := 49.579669; stNO_LENS[280].fHigh := 110.515509; 
    stNO_LENS[281].fEnergy := 8892.403578; stNO_LENS[281].fLow := 49.370931; stNO_LENS[281].fHigh := 110.071554; 
    stNO_LENS[282].fEnergy := 8910.206181; stNO_LENS[282].fLow := 49.163083; stNO_LENS[282].fHigh := 109.629572; 
    stNO_LENS[283].fEnergy := 8928.044426; stNO_LENS[283].fLow := 48.956123; stNO_LENS[283].fHigh := 109.189554; 
    stNO_LENS[284].fEnergy := 8945.918383; stNO_LENS[284].fLow := 48.750046; stNO_LENS[284].fHigh := 108.751491; 
    stNO_LENS[285].fEnergy := 8963.828123; stNO_LENS[285].fLow := 48.544850; stNO_LENS[285].fHigh := 108.315376; 
    stNO_LENS[286].fEnergy := 8981.773719; stNO_LENS[286].fLow := 48.340531; stNO_LENS[286].fHigh := 107.881198; 
    stNO_LENS[287].fEnergy := 8999.755242; stNO_LENS[287].fLow := 48.137087; stNO_LENS[287].fHigh := 107.448951; 
    stNO_LENS[288].fEnergy := 9017.772764; stNO_LENS[288].fLow := 47.934513; stNO_LENS[288].fHigh := 107.018624; 
    stNO_LENS[289].fEnergy := 9035.826357; stNO_LENS[289].fLow := 47.732807; stNO_LENS[289].fHigh := 106.590209; 
    stNO_LENS[290].fEnergy := 9053.916094; stNO_LENS[290].fLow := 47.531965; stNO_LENS[290].fHigh := 106.163697; 
    stNO_LENS[291].fEnergy := 9072.042046; stNO_LENS[291].fLow := 47.331984; stNO_LENS[291].fHigh := 105.739080; 
    stNO_LENS[292].fEnergy := 9090.204286; stNO_LENS[292].fLow := 47.132860; stNO_LENS[292].fHigh := 105.316349; 
    stNO_LENS[293].fEnergy := 9108.402887; stNO_LENS[293].fLow := 46.934592; stNO_LENS[293].fHigh := 104.895495; 
    stNO_LENS[294].fEnergy := 9126.637922; stNO_LENS[294].fLow := 46.737174; stNO_LENS[294].fHigh := 104.476508; 
    stNO_LENS[295].fEnergy := 9144.909463; stNO_LENS[295].fLow := 46.540605; stNO_LENS[295].fHigh := 104.059382; 
    stNO_LENS[296].fEnergy := 9163.217584; stNO_LENS[296].fLow := 46.344880; stNO_LENS[296].fHigh := 103.644106; 
    stNO_LENS[297].fEnergy := 9181.562358; stNO_LENS[297].fLow := 46.149998; stNO_LENS[297].fHigh := 103.230671; 
    stNO_LENS[298].fEnergy := 9199.943858; stNO_LENS[298].fLow := 45.955953; stNO_LENS[298].fHigh := 102.819070; 
    stNO_LENS[299].fEnergy := 9218.362158; stNO_LENS[299].fLow := 45.762744; stNO_LENS[299].fHigh := 102.409293; 
    stNO_LENS[300].fEnergy := 9236.817331; stNO_LENS[300].fLow := 45.570367; stNO_LENS[300].fHigh := 102.001331; 
    stNO_LENS[301].fEnergy := 9255.309452; stNO_LENS[301].fLow := 45.378819; stNO_LENS[301].fHigh := 101.595176; 
    stNO_LENS[302].fEnergy := 9273.838594; stNO_LENS[302].fLow := 45.188096; stNO_LENS[302].fHigh := 101.190820; 
    stNO_LENS[303].fEnergy := 9292.404831; stNO_LENS[303].fLow := 44.998196; stNO_LENS[303].fHigh := 100.788252; 
    stNO_LENS[304].fEnergy := 9311.008238; stNO_LENS[304].fLow := 44.809116; stNO_LENS[304].fHigh := 100.387465; 
    stNO_LENS[305].fEnergy := 9329.648889; stNO_LENS[305].fLow := 44.620851; stNO_LENS[305].fHigh := 99.988451; 
    stNO_LENS[306].fEnergy := 9348.326858; stNO_LENS[306].fLow := 44.433400; stNO_LENS[306].fHigh := 99.591199; 
    stNO_LENS[307].fEnergy := 9367.042221; stNO_LENS[307].fLow := 44.246758; stNO_LENS[307].fHigh := 99.195703; 
    stNO_LENS[308].fEnergy := 9385.795052; stNO_LENS[308].fLow := 44.060924; stNO_LENS[308].fHigh := 98.801953; 
    stNO_LENS[309].fEnergy := 9404.585426; stNO_LENS[309].fLow := 43.875892; stNO_LENS[309].fHigh := 98.409940; 
    stNO_LENS[310].fEnergy := 9423.413419; stNO_LENS[310].fLow := 43.691662; stNO_LENS[310].fHigh := 98.019657; 
    stNO_LENS[311].fEnergy := 9442.279105; stNO_LENS[311].fLow := 43.508228; stNO_LENS[311].fHigh := 97.631095; 
    stNO_LENS[312].fEnergy := 9461.182561; stNO_LENS[312].fLow := 43.325589; stNO_LENS[312].fHigh := 97.244245; 
    stNO_LENS[313].fEnergy := 9480.123861; stNO_LENS[313].fLow := 43.143741; stNO_LENS[313].fHigh := 96.859099; 
    stNO_LENS[314].fEnergy := 9499.103081; stNO_LENS[314].fLow := 42.962681; stNO_LENS[314].fHigh := 96.475649; 
    stNO_LENS[315].fEnergy := 9518.120298; stNO_LENS[315].fLow := 42.782406; stNO_LENS[315].fHigh := 96.093886; 
    stNO_LENS[316].fEnergy := 9537.175588; stNO_LENS[316].fLow := 42.602913; stNO_LENS[316].fHigh := 95.713802; 
    stNO_LENS[317].fEnergy := 9556.269026; stNO_LENS[317].fLow := 42.424199; stNO_LENS[317].fHigh := 95.335389; 
    stNO_LENS[318].fEnergy := 9575.400690; stNO_LENS[318].fLow := 42.246260; stNO_LENS[318].fHigh := 94.958639; 
    stNO_LENS[319].fEnergy := 9594.570654; stNO_LENS[319].fLow := 42.069094; stNO_LENS[319].fHigh := 94.583544; 
    stNO_LENS[320].fEnergy := 9613.778998; stNO_LENS[320].fLow := 41.892698; stNO_LENS[320].fHigh := 94.210095; 
    stNO_LENS[321].fEnergy := 9633.025796; stNO_LENS[321].fLow := 41.717068; stNO_LENS[321].fHigh := 93.838284; 
    stNO_LENS[322].fEnergy := 9652.311127; stNO_LENS[322].fLow := 41.542202; stNO_LENS[322].fHigh := 93.468104; 
    stNO_LENS[323].fEnergy := 9671.635066; stNO_LENS[323].fLow := 41.368096; stNO_LENS[323].fHigh := 93.099547; 
    stNO_LENS[324].fEnergy := 9690.997693; stNO_LENS[324].fLow := 41.194747; stNO_LENS[324].fHigh := 92.732605; 
    stNO_LENS[325].fEnergy := 9710.399083; stNO_LENS[325].fLow := 41.022153; stNO_LENS[325].fHigh := 92.367269; 
    stNO_LENS[326].fEnergy := 9729.839315; stNO_LENS[326].fLow := 40.850310; stNO_LENS[326].fHigh := 92.003533; 
    stNO_LENS[327].fEnergy := 9749.318466; stNO_LENS[327].fLow := 40.679216; stNO_LENS[327].fHigh := 91.641387; 
    stNO_LENS[328].fEnergy := 9768.836615; stNO_LENS[328].fLow := 40.508867; stNO_LENS[328].fHigh := 91.280826; 
    stNO_LENS[329].fEnergy := 9788.393839; stNO_LENS[329].fLow := 40.339260; stNO_LENS[329].fHigh := 90.921840; 
    stNO_LENS[330].fEnergy := 9807.990216; stNO_LENS[330].fLow := 40.170393; stNO_LENS[330].fHigh := 90.564423; 
    stNO_LENS[331].fEnergy := 9827.625826; stNO_LENS[331].fLow := 40.002262; stNO_LENS[331].fHigh := 90.208567; 
    stNO_LENS[332].fEnergy := 9847.300746; stNO_LENS[332].fLow := 39.834865; stNO_LENS[332].fHigh := 89.854264; 
    stNO_LENS[333].fEnergy := 9867.015055; stNO_LENS[333].fLow := 39.668198; stNO_LENS[333].fHigh := 89.501508; 
    stNO_LENS[334].fEnergy := 9886.768832; stNO_LENS[334].fLow := 39.502259; stNO_LENS[334].fHigh := 89.150289; 
    stNO_LENS[335].fEnergy := 9906.562157; stNO_LENS[335].fLow := 39.337044; stNO_LENS[335].fHigh := 88.800602; 
    stNO_LENS[336].fEnergy := 9926.395107; stNO_LENS[336].fLow := 39.172551; stNO_LENS[336].fHigh := 88.452439; 
    stNO_LENS[337].fEnergy := 9946.267764; stNO_LENS[337].fLow := 39.008777; stNO_LENS[337].fHigh := 88.105793; 
    stNO_LENS[338].fEnergy := 9966.180205; stNO_LENS[338].fLow := 38.845718; stNO_LENS[338].fHigh := 87.760656; 
    stNO_LENS[339].fEnergy := 9986.132511; stNO_LENS[339].fLow := 38.683373; stNO_LENS[339].fHigh := 87.417021; 
    stNO_LENS[340].fEnergy := 10006.124762; stNO_LENS[340].fLow := 38.521737; stNO_LENS[340].fHigh := 87.074881; 
    stNO_LENS[341].fEnergy := 10026.157037; stNO_LENS[341].fLow := 38.360808; stNO_LENS[341].fHigh := 86.734230; 
    stNO_LENS[342].fEnergy := 10046.229416; stNO_LENS[342].fLow := 38.200584; stNO_LENS[342].fHigh := 86.395060; 
    stNO_LENS[343].fEnergy := 10066.341981; stNO_LENS[343].fLow := 38.041061; stNO_LENS[343].fHigh := 86.057364; 
    stNO_LENS[344].fEnergy := 10086.494811; stNO_LENS[344].fLow := 37.882236; stNO_LENS[344].fHigh := 85.721135; 
    stNO_LENS[345].fEnergy := 10106.687987; stNO_LENS[345].fLow := 37.724107; stNO_LENS[345].fHigh := 85.386367; 
    stNO_LENS[346].fEnergy := 10126.921590; stNO_LENS[346].fLow := 37.566671; stNO_LENS[346].fHigh := 85.053052; 
    stNO_LENS[347].fEnergy := 10147.195701; stNO_LENS[347].fLow := 37.409925; stNO_LENS[347].fHigh := 84.721184; 
    stNO_LENS[348].fEnergy := 10167.510400; stNO_LENS[348].fLow := 37.253865; stNO_LENS[348].fHigh := 84.390755; 
    stNO_LENS[349].fEnergy := 10187.865769; stNO_LENS[349].fLow := 37.098490; stNO_LENS[349].fHigh := 84.061760; 
    stNO_LENS[350].fEnergy := 10208.261890; stNO_LENS[350].fLow := 36.943796; stNO_LENS[350].fHigh := 83.734192; 
    stNO_LENS[351].fEnergy := 10228.698844; stNO_LENS[351].fLow := 36.789781; stNO_LENS[351].fHigh := 83.408044; 
    stNO_LENS[352].fEnergy := 10249.176713; stNO_LENS[352].fLow := 36.636441; stNO_LENS[352].fHigh := 83.083309; 
    stNO_LENS[353].fEnergy := 10269.695578; stNO_LENS[353].fLow := 36.483775; stNO_LENS[353].fHigh := 82.759981; 
    stNO_LENS[354].fEnergy := 10290.255523; stNO_LENS[354].fLow := 36.331778; stNO_LENS[354].fHigh := 82.438054; 
    stNO_LENS[355].fEnergy := 10310.856628; stNO_LENS[355].fLow := 36.180449; stNO_LENS[355].fHigh := 82.117520; 
    stNO_LENS[356].fEnergy := 10331.498977; stNO_LENS[356].fLow := 36.029784; stNO_LENS[356].fHigh := 81.798374; 
    stNO_LENS[357].fEnergy := 10352.182651; stNO_LENS[357].fLow := 35.879782; stNO_LENS[357].fHigh := 81.480609; 
    stNO_LENS[358].fEnergy := 10372.907735; stNO_LENS[358].fLow := 35.730438; stNO_LENS[358].fHigh := 81.164218; 
    stNO_LENS[359].fEnergy := 10393.674310; stNO_LENS[359].fLow := 35.581750; stNO_LENS[359].fHigh := 80.849196; 
    stNO_LENS[360].fEnergy := 10414.482460; stNO_LENS[360].fLow := 35.433716; stNO_LENS[360].fHigh := 80.535536; 
    stNO_LENS[361].fEnergy := 10435.332268; stNO_LENS[361].fLow := 35.286333; stNO_LENS[361].fHigh := 80.223232; 
    stNO_LENS[362].fEnergy := 10456.223817; stNO_LENS[362].fLow := 35.139598; stNO_LENS[362].fHigh := 79.912277; 
    stNO_LENS[363].fEnergy := 10477.157191; stNO_LENS[363].fLow := 34.993508; stNO_LENS[363].fHigh := 79.602666; 
    stNO_LENS[364].fEnergy := 10498.132473; stNO_LENS[364].fLow := 34.848061; stNO_LENS[364].fHigh := 79.294391; 
    stNO_LENS[365].fEnergy := 10519.149749; stNO_LENS[365].fLow := 34.703254; stNO_LENS[365].fHigh := 78.987448; 
    stNO_LENS[366].fEnergy := 10540.209100; stNO_LENS[366].fLow := 34.559084; stNO_LENS[366].fHigh := 78.681829; 
    stNO_LENS[367].fEnergy := 10561.310613; stNO_LENS[367].fLow := 34.415549; stNO_LENS[367].fHigh := 78.377529; 
    stNO_LENS[368].fEnergy := 10582.454371; stNO_LENS[368].fLow := 34.272645; stNO_LENS[368].fHigh := 78.074542; 
    stNO_LENS[369].fEnergy := 10603.640459; stNO_LENS[369].fLow := 34.130371; stNO_LENS[369].fHigh := 77.772861; 
    stNO_LENS[370].fEnergy := 10624.868961; stNO_LENS[370].fLow := 33.988723; stNO_LENS[370].fHigh := 77.472481; 
    stNO_LENS[371].fEnergy := 10646.139963; stNO_LENS[371].fLow := 33.847699; stNO_LENS[371].fHigh := 77.173395; 
    stNO_LENS[372].fEnergy := 10667.453549; stNO_LENS[372].fLow := 33.707297; stNO_LENS[372].fHigh := 76.875597; 
    stNO_LENS[373].fEnergy := 10688.809806; stNO_LENS[373].fLow := 33.567513; stNO_LENS[373].fHigh := 76.579082; 
    stNO_LENS[374].fEnergy := 10710.208817; stNO_LENS[374].fLow := 33.428345; stNO_LENS[374].fHigh := 76.283844; 
    stNO_LENS[375].fEnergy := 10731.650669; stNO_LENS[375].fLow := 33.289790; stNO_LENS[375].fHigh := 75.989875; 
    stNO_LENS[376].fEnergy := 10753.135448; stNO_LENS[376].fLow := 33.151846; stNO_LENS[376].fHigh := 75.697171; 
    stNO_LENS[377].fEnergy := 10774.663240; stNO_LENS[377].fLow := 33.014510; stNO_LENS[377].fHigh := 75.405726; 
    stNO_LENS[378].fEnergy := 10796.234130; stNO_LENS[378].fLow := 32.877780; stNO_LENS[378].fHigh := 75.115533; 
    stNO_LENS[379].fEnergy := 10817.848205; stNO_LENS[379].fLow := 32.741653; stNO_LENS[379].fHigh := 74.826587; 
    stNO_LENS[380].fEnergy := 10839.505552; stNO_LENS[380].fLow := 32.606126; stNO_LENS[380].fHigh := 74.538882; 
    stNO_LENS[381].fEnergy := 10861.206256; stNO_LENS[381].fLow := 32.471197; stNO_LENS[381].fHigh := 74.252411; 
    stNO_LENS[382].fEnergy := 10882.950406; stNO_LENS[382].fLow := 32.336863; stNO_LENS[382].fHigh := 73.967170; 
    stNO_LENS[383].fEnergy := 10904.738087; stNO_LENS[383].fLow := 32.203122; stNO_LENS[383].fHigh := 73.683151; 
    stNO_LENS[384].fEnergy := 10926.569387; stNO_LENS[384].fLow := 32.069971; stNO_LENS[384].fHigh := 73.400349; 
    stNO_LENS[385].fEnergy := 10948.444394; stNO_LENS[385].fLow := 31.937407; stNO_LENS[385].fHigh := 73.118758; 
    stNO_LENS[386].fEnergy := 10970.363194; stNO_LENS[386].fLow := 31.805429; stNO_LENS[386].fHigh := 72.838373; 
    stNO_LENS[387].fEnergy := 10992.325876; stNO_LENS[387].fLow := 31.674033; stNO_LENS[387].fHigh := 72.559186; 
    stNO_LENS[388].fEnergy := 11014.332527; stNO_LENS[388].fLow := 31.543218; stNO_LENS[388].fHigh := 72.281193; 
    stNO_LENS[389].fEnergy := 11036.383235; stNO_LENS[389].fLow := 31.412979; stNO_LENS[389].fHigh := 72.004387; 
    stNO_LENS[390].fEnergy := 11058.478089; stNO_LENS[390].fLow := 31.283316; stNO_LENS[390].fHigh := 71.728763; 
    stNO_LENS[391].fEnergy := 11080.617177; stNO_LENS[391].fLow := 31.154226; stNO_LENS[391].fHigh := 71.454314; 
    stNO_LENS[392].fEnergy := 11102.800587; stNO_LENS[392].fLow := 31.025705; stNO_LENS[392].fHigh := 71.181035; 
    stNO_LENS[393].fEnergy := 11125.028409; stNO_LENS[393].fLow := 30.897753; stNO_LENS[393].fHigh := 70.908919; 
    stNO_LENS[394].fEnergy := 11147.300731; stNO_LENS[394].fLow := 30.770365; stNO_LENS[394].fHigh := 70.637961; 
    stNO_LENS[395].fEnergy := 11169.617642; stNO_LENS[395].fLow := 30.643540; stNO_LENS[395].fHigh := 70.368154; 
    stNO_LENS[396].fEnergy := 11191.979231; stNO_LENS[396].fLow := 30.517276; stNO_LENS[396].fHigh := 70.099493; 
    stNO_LENS[397].fEnergy := 11214.385588; stNO_LENS[397].fLow := 30.391569; stNO_LENS[397].fHigh := 69.831971; 
    stNO_LENS[398].fEnergy := 11236.836803; stNO_LENS[398].fLow := 30.266418; stNO_LENS[398].fHigh := 69.565583; 
    stNO_LENS[399].fEnergy := 11259.332966; stNO_LENS[399].fLow := 30.141819; stNO_LENS[399].fHigh := 69.300322; 
    stNO_LENS[400].fEnergy := 11281.874165; stNO_LENS[400].fLow := 30.017771; stNO_LENS[400].fHigh := 69.036182; 
    stNO_LENS[401].fEnergy := 11304.460492; stNO_LENS[401].fLow := 29.894272; stNO_LENS[401].fHigh := 68.773157; 
    stNO_LENS[402].fEnergy := 11327.092037; stNO_LENS[402].fLow := 29.771318; stNO_LENS[402].fHigh := 68.511241; 
    stNO_LENS[403].fEnergy := 11349.768891; stNO_LENS[403].fLow := 29.648908; stNO_LENS[403].fHigh := 68.250428; 
    stNO_LENS[404].fEnergy := 11372.491143; stNO_LENS[404].fLow := 29.527038; stNO_LENS[404].fHigh := 67.990712; 
    stNO_LENS[405].fEnergy := 11395.258886; stNO_LENS[405].fLow := 29.405707; stNO_LENS[405].fHigh := 67.732085; 
    stNO_LENS[406].fEnergy := 11418.072209; stNO_LENS[406].fLow := 29.284913; stNO_LENS[406].fHigh := 67.474543; 
    stNO_LENS[407].fEnergy := 11440.931205; stNO_LENS[407].fLow := 29.164652; stNO_LENS[407].fHigh := 67.218079; 
    stNO_LENS[408].fEnergy := 11463.835964; stNO_LENS[408].fLow := 29.044924; stNO_LENS[408].fHigh := 66.962686; 
    stNO_LENS[409].fEnergy := 11486.786579; stNO_LENS[409].fLow := 28.925724; stNO_LENS[409].fHigh := 66.708358; 
    stNO_LENS[410].fEnergy := 11509.783141; stNO_LENS[410].fLow := 28.807051; stNO_LENS[410].fHigh := 66.455089; 
    stNO_LENS[411].fEnergy := 11532.825743; stNO_LENS[411].fLow := 28.688903; stNO_LENS[411].fHigh := 66.202873; 
    stNO_LENS[412].fEnergy := 11555.914475; stNO_LENS[412].fLow := 28.571278; stNO_LENS[412].fHigh := 65.951702; 
    stNO_LENS[413].fEnergy := 11579.049431; stNO_LENS[413].fLow := 28.454172; stNO_LENS[413].fHigh := 65.701570; 
    stNO_LENS[414].fEnergy := 11602.230704; stNO_LENS[414].fLow := 28.337584; stNO_LENS[414].fHigh := 65.452471; 
    stNO_LENS[415].fEnergy := 11625.458385; stNO_LENS[415].fLow := 28.221511; stNO_LENS[415].fHigh := 65.204398; 
    stNO_LENS[416].fEnergy := 11648.732568; stNO_LENS[416].fLow := 28.105952; stNO_LENS[416].fHigh := 64.957344; 
    stNO_LENS[417].fEnergy := 11672.053346; stNO_LENS[417].fLow := 27.990903; stNO_LENS[417].fHigh := 64.711303; 
    stNO_LENS[418].fEnergy := 11695.420813; stNO_LENS[418].fLow := 27.876363; stNO_LENS[418].fHigh := 64.466269; 
    stNO_LENS[419].fEnergy := 11718.835061; stNO_LENS[419].fLow := 27.762330; stNO_LENS[419].fHigh := 64.222233; 
    stNO_LENS[420].fEnergy := 11742.296184; stNO_LENS[420].fLow := 27.648801; stNO_LENS[420].fHigh := 63.979190; 
    stNO_LENS[421].fEnergy := 11765.804277; stNO_LENS[421].fLow := 27.535773; stNO_LENS[421].fHigh := 63.737133; 
    stNO_LENS[422].fEnergy := 11789.359433; stNO_LENS[422].fLow := 27.423245; stNO_LENS[422].fHigh := 63.496054; 
    stNO_LENS[423].fEnergy := 11812.961746; stNO_LENS[423].fLow := 27.311215; stNO_LENS[423].fHigh := 63.255947; 
    stNO_LENS[424].fEnergy := 11836.611311; stNO_LENS[424].fLow := 27.199680; stNO_LENS[424].fHigh := 63.016804; 
    stNO_LENS[425].fEnergy := 11860.308223; stNO_LENS[425].fLow := 27.088638; stNO_LENS[425].fHigh := 62.778619; 
    stNO_LENS[426].fEnergy := 11884.052576; stNO_LENS[426].fLow := 26.978087; stNO_LENS[426].fHigh := 62.541384; 
    stNO_LENS[427].fEnergy := 11907.844465; stNO_LENS[427].fLow := 26.868024; stNO_LENS[427].fHigh := 62.305093; 
    stNO_LENS[428].fEnergy := 11931.683985; stNO_LENS[428].fLow := 26.758448; stNO_LENS[428].fHigh := 62.069737; 
    stNO_LENS[429].fEnergy := 11955.571233; stNO_LENS[429].fLow := 26.649356; stNO_LENS[429].fHigh := 61.835309; 
    stNO_LENS[430].fEnergy := 11979.506302; stNO_LENS[430].fLow := 26.540747; stNO_LENS[430].fHigh := 61.601803; 
    stNO_LENS[431].fEnergy := 12003.489290; stNO_LENS[431].fLow := 26.432617; stNO_LENS[431].fHigh := 61.369210; 
    stNO_LENS[432].fEnergy := 12027.520291; stNO_LENS[432].fLow := 26.324966; stNO_LENS[432].fHigh := 61.137524; 
    stNO_LENS[433].fEnergy := 12051.599403; stNO_LENS[433].fLow := 26.217790; stNO_LENS[433].fHigh := 60.906736; 
    stNO_LENS[434].fEnergy := 12075.726721; stNO_LENS[434].fLow := 26.111087; stNO_LENS[434].fHigh := 60.676839; 
    stNO_LENS[435].fEnergy := 12099.902342; stNO_LENS[435].fLow := 26.004856; stNO_LENS[435].fHigh := 60.447825; 
    stNO_LENS[436].fEnergy := 12124.126363; stNO_LENS[436].fLow := 25.899095; stNO_LENS[436].fHigh := 60.219687; 
    stNO_LENS[437].fEnergy := 12148.398880; stNO_LENS[437].fLow := 25.793801; stNO_LENS[437].fHigh := 59.992415; 
    stNO_LENS[438].fEnergy := 12172.719991; stNO_LENS[438].fLow := 25.688971; stNO_LENS[438].fHigh := 59.766004; 
    stNO_LENS[439].fEnergy := 12197.089792; stNO_LENS[439].fLow := 25.584605; stNO_LENS[439].fHigh := 59.540444; 
    stNO_LENS[440].fEnergy := 12221.508382; stNO_LENS[440].fLow := 25.480700; stNO_LENS[440].fHigh := 59.315728; 
    stNO_LENS[441].fEnergy := 12245.975858; stNO_LENS[441].fLow := 25.377254; stNO_LENS[441].fHigh := 59.091847; 
    stNO_LENS[442].fEnergy := 12270.492318; stNO_LENS[442].fLow := 25.274265; stNO_LENS[442].fHigh := 58.868793; 
    stNO_LENS[443].fEnergy := 12295.057860; stNO_LENS[443].fLow := 25.171730; stNO_LENS[443].fHigh := 58.646558; 
    stNO_LENS[444].fEnergy := 12319.672583; stNO_LENS[444].fLow := 25.069649; stNO_LENS[444].fHigh := 58.425133; 
    stNO_LENS[445].fEnergy := 12344.336584; stNO_LENS[445].fLow := 24.968018; stNO_LENS[445].fHigh := 58.204510; 
    stNO_LENS[446].fEnergy := 12369.049962; stNO_LENS[446].fLow := 24.866835; stNO_LENS[446].fHigh := 57.984681; 
    stNO_LENS[447].fEnergy := 12393.812816; stNO_LENS[447].fLow := 24.766100; stNO_LENS[447].fHigh := 57.765636; 
    stNO_LENS[448].fEnergy := 12418.625246; stNO_LENS[448].fLow := 24.665808; stNO_LENS[448].fHigh := 57.547368; 
    stNO_LENS[449].fEnergy := 12443.487350; stNO_LENS[449].fLow := 24.565960; stNO_LENS[449].fHigh := 57.329867; 
    stNO_LENS[450].fEnergy := 12468.399229; stNO_LENS[450].fLow := 24.466552; stNO_LENS[450].fHigh := 57.113125; 
    stNO_LENS[451].fEnergy := 12493.360981; stNO_LENS[451].fLow := 24.367583; stNO_LENS[451].fHigh := 56.897132; 
    stNO_LENS[452].fEnergy := 12518.372706; stNO_LENS[452].fLow := 24.269051; stNO_LENS[452].fHigh := 56.681879; 
    stNO_LENS[453].fEnergy := 12543.434505; stNO_LENS[453].fLow := 24.170953; stNO_LENS[453].fHigh := 56.467358; 
    stNO_LENS[454].fEnergy := 12568.546477; stNO_LENS[454].fLow := 24.073288; stNO_LENS[454].fHigh := 56.253559; 
    stNO_LENS[455].fEnergy := 12593.708724; stNO_LENS[455].fLow := 23.976053; stNO_LENS[455].fHigh := 56.040473; 
    stNO_LENS[456].fEnergy := 12618.921346; stNO_LENS[456].fLow := 23.879248; stNO_LENS[456].fHigh := 55.828091; 
    stNO_LENS[457].fEnergy := 12644.184443; stNO_LENS[457].fLow := 23.782869; stNO_LENS[457].fHigh := 55.616402; 
    stNO_LENS[458].fEnergy := 12669.498117; stNO_LENS[458].fLow := 23.686915; stNO_LENS[458].fHigh := 55.405399; 
    stNO_LENS[459].fEnergy := 12694.862470; stNO_LENS[459].fLow := 23.591384; stNO_LENS[459].fHigh := 55.195070; 
    stNO_LENS[460].fEnergy := 12720.277601; stNO_LENS[460].fLow := 23.496274; stNO_LENS[460].fHigh := 54.954308; 
    stNO_LENS[461].fEnergy := 12745.743614; stNO_LENS[461].fLow := 23.401583; stNO_LENS[461].fHigh := 54.755484; 
    stNO_LENS[462].fEnergy := 12771.260610; stNO_LENS[462].fLow := 23.307310; stNO_LENS[462].fHigh := 54.556824; 
    stNO_LENS[463].fEnergy := 12796.828690; stNO_LENS[463].fLow := 23.213452; stNO_LENS[463].fHigh := 54.358351; 
    stNO_LENS[464].fEnergy := 12822.447958; stNO_LENS[464].fLow := 23.120007; stNO_LENS[464].fHigh := 54.160086; 
    stNO_LENS[465].fEnergy := 12848.118516; stNO_LENS[465].fLow := 23.026974; stNO_LENS[465].fHigh := 53.962051; 
    stNO_LENS[466].fEnergy := 12873.840467; stNO_LENS[466].fLow := 22.934350; stNO_LENS[466].fHigh := 53.764265; 
    stNO_LENS[467].fEnergy := 12899.613913; stNO_LENS[467].fLow := 22.842135; stNO_LENS[467].fHigh := 53.566749; 
    stNO_LENS[468].fEnergy := 12925.438957; stNO_LENS[468].fLow := 22.750325; stNO_LENS[468].fHigh := 53.369520; 
    stNO_LENS[469].fEnergy := 12951.315703; stNO_LENS[469].fLow := 22.658919; stNO_LENS[469].fHigh := 53.172597; 
    stNO_LENS[470].fEnergy := 12977.244254; stNO_LENS[470].fLow := 22.567916; stNO_LENS[470].fHigh := 52.975997; 
    stNO_LENS[471].fEnergy := 13003.224714; stNO_LENS[471].fLow := 22.477313; stNO_LENS[471].fHigh := 52.779737; 
    stNO_LENS[472].fEnergy := 13029.257188; stNO_LENS[472].fLow := 22.387108; stNO_LENS[472].fHigh := 52.583832; 
    stNO_LENS[473].fEnergy := 13055.341778; stNO_LENS[473].fLow := 22.297301; stNO_LENS[473].fHigh := 52.388298; 
    stNO_LENS[474].fEnergy := 13081.478590; stNO_LENS[474].fLow := 22.207888; stNO_LENS[474].fHigh := 52.193149; 
    stNO_LENS[475].fEnergy := 13107.667727; stNO_LENS[475].fLow := 22.118868; stNO_LENS[475].fHigh := 51.998399; 
    stNO_LENS[476].fEnergy := 13133.909296; stNO_LENS[476].fLow := 22.030240; stNO_LENS[476].fHigh := 51.804063; 
    stNO_LENS[477].fEnergy := 13160.203399; stNO_LENS[477].fLow := 21.942001; stNO_LENS[477].fHigh := 51.610151; 
    stNO_LENS[478].fEnergy := 13186.550144; stNO_LENS[478].fLow := 21.854150; stNO_LENS[478].fHigh := 51.416677; 
    stNO_LENS[479].fEnergy := 13212.949635; stNO_LENS[479].fLow := 21.766685; stNO_LENS[479].fHigh := 51.223653; 
    stNO_LENS[480].fEnergy := 13239.401978; stNO_LENS[480].fLow := 21.679604; stNO_LENS[480].fHigh := 51.031089; 
    stNO_LENS[481].fEnergy := 13265.907278; stNO_LENS[481].fLow := 21.592905; stNO_LENS[481].fHigh := 50.838996; 
    stNO_LENS[482].fEnergy := 13292.465642; stNO_LENS[482].fLow := 21.506588; stNO_LENS[482].fHigh := 50.647384; 
    stNO_LENS[483].fEnergy := 13319.077176; stNO_LENS[483].fLow := 21.420649; stNO_LENS[483].fHigh := 50.456262; 
    stNO_LENS[484].fEnergy := 13345.741987; stNO_LENS[484].fLow := 21.335087; stNO_LENS[484].fHigh := 50.265640; 
    stNO_LENS[485].fEnergy := 13372.460180; stNO_LENS[485].fLow := 21.249901; stNO_LENS[485].fHigh := 50.075527; 
    stNO_LENS[486].fEnergy := 13399.231863; stNO_LENS[486].fLow := 21.165088; stNO_LENS[486].fHigh := 49.885929; 
    stNO_LENS[487].fEnergy := 13426.057143; stNO_LENS[487].fLow := 21.080647; stNO_LENS[487].fHigh := 49.696856; 
    stNO_LENS[488].fEnergy := 13452.936127; stNO_LENS[488].fLow := 20.996577; stNO_LENS[488].fHigh := 49.508314; 
    stNO_LENS[489].fEnergy := 13479.868924; stNO_LENS[489].fLow := 20.912875; stNO_LENS[489].fHigh := 49.320310; 
    stNO_LENS[490].fEnergy := 13506.855639; stNO_LENS[490].fLow := 20.829540; stNO_LENS[490].fHigh := 49.132851; 
    stNO_LENS[491].fEnergy := 13533.896382; stNO_LENS[491].fLow := 20.746570; stNO_LENS[491].fHigh := 48.945942; 
    stNO_LENS[492].fEnergy := 13560.991261; stNO_LENS[492].fLow := 20.663964; stNO_LENS[492].fHigh := 48.759590; 
    stNO_LENS[493].fEnergy := 13588.140383; stNO_LENS[493].fLow := 20.581719; stNO_LENS[493].fHigh := 48.573799; 
    stNO_LENS[494].fEnergy := 13615.343858; stNO_LENS[494].fLow := 20.499835; stNO_LENS[494].fHigh := 48.388575; 
    stNO_LENS[495].fEnergy := 13642.601795; stNO_LENS[495].fLow := 20.418309; stNO_LENS[495].fHigh := 48.203921; 
    stNO_LENS[496].fEnergy := 13669.914302; stNO_LENS[496].fLow := 20.337140; stNO_LENS[496].fHigh := 48.019843; 
    stNO_LENS[497].fEnergy := 13697.281489; stNO_LENS[497].fLow := 20.256326; stNO_LENS[497].fHigh := 47.836344; 
    stNO_LENS[498].fEnergy := 13724.703465; stNO_LENS[498].fLow := 20.175866; stNO_LENS[498].fHigh := 47.653428; 
    stNO_LENS[499].fEnergy := 13752.180339; stNO_LENS[499].fLow := 20.095757; stNO_LENS[499].fHigh := 47.471098; 
    stNO_LENS[500].fEnergy := 13779.712223; stNO_LENS[500].fLow := 20.015999; stNO_LENS[500].fHigh := 47.289358; 
    stNO_LENS[501].fEnergy := 13807.299225; stNO_LENS[501].fLow := 19.936589; stNO_LENS[501].fHigh := 47.108209; 
    stNO_LENS[502].fEnergy := 13834.941456; stNO_LENS[502].fLow := 19.857526; stNO_LENS[502].fHigh := 46.927654; 
    stNO_LENS[503].fEnergy := 13862.639028; stNO_LENS[503].fLow := 19.778809; stNO_LENS[503].fHigh := 46.747696; 
    stNO_LENS[504].fEnergy := 13890.392049; stNO_LENS[504].fLow := 19.700436; stNO_LENS[504].fHigh := 46.568337; 
    stNO_LENS[505].fEnergy := 13918.200633; stNO_LENS[505].fLow := 19.622404; stNO_LENS[505].fHigh := 46.389577; 
    stNO_LENS[506].fEnergy := 13946.064889; stNO_LENS[506].fLow := 19.544714; stNO_LENS[506].fHigh := 46.211420; 
    stNO_LENS[507].fEnergy := 13973.984929; stNO_LENS[507].fLow := 19.467362; stNO_LENS[507].fHigh := 46.033865; 
    stNO_LENS[508].fEnergy := 14001.960866; stNO_LENS[508].fLow := 19.390348; stNO_LENS[508].fHigh := 45.856914; 
    stNO_LENS[509].fEnergy := 14029.992810; stNO_LENS[509].fLow := 19.313670; stNO_LENS[509].fHigh := 45.680568; 
    stNO_LENS[510].fEnergy := 14058.080875; stNO_LENS[510].fLow := 19.237326; stNO_LENS[510].fHigh := 45.504828; 
    stNO_LENS[511].fEnergy := 14086.225171; stNO_LENS[511].fLow := 19.161315; stNO_LENS[511].fHigh := 45.329693; 
    stNO_LENS[512].fEnergy := 14114.425813; stNO_LENS[512].fLow := 19.085635; stNO_LENS[512].fHigh := 45.155164; 
    stNO_LENS[513].fEnergy := 14142.682912; stNO_LENS[513].fLow := 19.010285; stNO_LENS[513].fHigh := 44.981241; 
    stNO_LENS[514].fEnergy := 14170.996582; stNO_LENS[514].fLow := 18.935263; stNO_LENS[514].fHigh := 44.807925; 
    stNO_LENS[515].fEnergy := 14199.366936; stNO_LENS[515].fLow := 18.860567; stNO_LENS[515].fHigh := 44.635214; 
    stNO_LENS[516].fEnergy := 14227.794088; stNO_LENS[516].fLow := 18.786197; stNO_LENS[516].fHigh := 44.463109; 
    stNO_LENS[517].fEnergy := 14256.278151; stNO_LENS[517].fLow := 18.712150; stNO_LENS[517].fHigh := 44.291608; 
    stNO_LENS[518].fEnergy := 14284.819238; stNO_LENS[518].fLow := 18.638426; stNO_LENS[518].fHigh := 44.120712; 
    stNO_LENS[519].fEnergy := 14313.417466; stNO_LENS[519].fLow := 18.565022; stNO_LENS[519].fHigh := 43.950419; 
    stNO_LENS[520].fEnergy := 14342.072946; stNO_LENS[520].fLow := 18.491937; stNO_LENS[520].fHigh := 43.780728; 
    stNO_LENS[521].fEnergy := 14370.785796; stNO_LENS[521].fLow := 18.419169; stNO_LENS[521].fHigh := 43.611638; 
    stNO_LENS[522].fEnergy := 14399.556128; stNO_LENS[522].fLow := 18.346718; stNO_LENS[522].fHigh := 43.443149; 
    stNO_LENS[523].fEnergy := 14428.384059; stNO_LENS[523].fLow := 18.274581; stNO_LENS[523].fHigh := 43.275258; 
    stNO_LENS[524].fEnergy := 14457.269703; stNO_LENS[524].fLow := 18.202758; stNO_LENS[524].fHigh := 43.107965; 
    stNO_LENS[525].fEnergy := 14486.213176; stNO_LENS[525].fLow := 18.131246; stNO_LENS[525].fHigh := 42.941268; 
    stNO_LENS[526].fEnergy := 14515.214594; stNO_LENS[526].fLow := 18.060045; stNO_LENS[526].fHigh := 42.775165; 
    stNO_LENS[527].fEnergy := 14544.274073; stNO_LENS[527].fLow := 17.989152; stNO_LENS[527].fHigh := 42.609655; 
    stNO_LENS[528].fEnergy := 14573.391729; stNO_LENS[528].fLow := 17.918567; stNO_LENS[528].fHigh := 42.444736; 
    stNO_LENS[529].fEnergy := 14602.567679; stNO_LENS[529].fLow := 17.848288; stNO_LENS[529].fHigh := 42.280406; 
    stNO_LENS[530].fEnergy := 14631.802039; stNO_LENS[530].fLow := 17.778313; stNO_LENS[530].fHigh := 42.116663; 
    stNO_LENS[531].fEnergy := 14661.094926; stNO_LENS[531].fLow := 17.708641; stNO_LENS[531].fHigh := 41.953505; 
    stNO_LENS[532].fEnergy := 14690.446458; stNO_LENS[532].fLow := 17.639271; stNO_LENS[532].fHigh := 41.790930; 
    stNO_LENS[533].fEnergy := 14719.856751; stNO_LENS[533].fLow := 17.570201; stNO_LENS[533].fHigh := 41.628937; 
    stNO_LENS[534].fEnergy := 14749.325924; stNO_LENS[534].fLow := 17.501430; stNO_LENS[534].fHigh := 41.467523; 
    stNO_LENS[535].fEnergy := 14778.854094; stNO_LENS[535].fLow := 17.432956; stNO_LENS[535].fHigh := 41.306685; 
    stNO_LENS[536].fEnergy := 14808.441380; stNO_LENS[536].fLow := 17.364779; stNO_LENS[536].fHigh := 41.146422; 
    stNO_LENS[537].fEnergy := 14838.087899; stNO_LENS[537].fLow := 17.296896; stNO_LENS[537].fHigh := 40.986732; 
    stNO_LENS[538].fEnergy := 14867.793771; stNO_LENS[538].fLow := 17.229306; stNO_LENS[538].fHigh := 40.827612; 
    stNO_LENS[539].fEnergy := 14897.559114; stNO_LENS[539].fLow := 17.162008; stNO_LENS[539].fHigh := 40.669059; 
    stNO_LENS[540].fEnergy := 14927.384047; stNO_LENS[540].fLow := 17.095001; stNO_LENS[540].fHigh := 40.511072; 
    stNO_LENS[541].fEnergy := 14957.268690; stNO_LENS[541].fLow := 17.028283; stNO_LENS[541].fHigh := 40.353647; 
    stNO_LENS[542].fEnergy := 14987.213162; stNO_LENS[542].fLow := 16.961853; stNO_LENS[542].fHigh := 40.196784; 
    stNO_LENS[543].fEnergy := 15017.217582; stNO_LENS[543].fLow := 16.895709; stNO_LENS[543].fHigh := 40.040478; 
    stNO_LENS[544].fEnergy := 15047.282072; stNO_LENS[544].fLow := 16.829850; stNO_LENS[544].fHigh := 39.884729; 
    stNO_LENS[545].fEnergy := 15077.406751; stNO_LENS[545].fLow := 16.764275; stNO_LENS[545].fHigh := 39.729532; 
    stNO_LENS[546].fEnergy := 15107.591739; stNO_LENS[546].fLow := 16.698983; stNO_LENS[546].fHigh := 39.574887; 
    stNO_LENS[547].fEnergy := 15137.837158; stNO_LENS[547].fLow := 16.633972; stNO_LENS[547].fHigh := 39.420790; 
    stNO_LENS[548].fEnergy := 15168.143128; stNO_LENS[548].fLow := 16.569240; stNO_LENS[548].fHigh := 39.267238; 
    stNO_LENS[549].fEnergy := 15198.509771; stNO_LENS[549].fLow := 16.504787; stNO_LENS[549].fHigh := 39.114230; 
    stNO_LENS[550].fEnergy := 15228.937208; stNO_LENS[550].fLow := 16.440611; stNO_LENS[550].fHigh := 38.961763; 
    stNO_LENS[551].fEnergy := 15259.425560; stNO_LENS[551].fLow := 16.376711; stNO_LENS[551].fHigh := 38.809835; 
    stNO_LENS[552].fEnergy := 15289.974951; stNO_LENS[552].fLow := 16.313086; stNO_LENS[552].fHigh := 38.658443; 
    stNO_LENS[553].fEnergy := 15320.585501; stNO_LENS[553].fLow := 16.249734; stNO_LENS[553].fHigh := 38.507584; 
    stNO_LENS[554].fEnergy := 15351.257334; stNO_LENS[554].fLow := 16.186654; stNO_LENS[554].fHigh := 38.357256; 
    stNO_LENS[555].fEnergy := 15381.990571; stNO_LENS[555].fLow := 16.123844; stNO_LENS[555].fHigh := 38.207457; 
    stNO_LENS[556].fEnergy := 15412.785337; stNO_LENS[556].fLow := 16.061304; stNO_LENS[556].fHigh := 38.058184; 
    stNO_LENS[557].fEnergy := 15443.641754; stNO_LENS[557].fLow := 15.999032; stNO_LENS[557].fHigh := 37.909435; 
    stNO_LENS[558].fEnergy := 15474.559945; stNO_LENS[558].fLow := 15.937027; stNO_LENS[558].fHigh := 37.761208; 
    stNO_LENS[559].fEnergy := 15505.540035; stNO_LENS[559].fLow := 15.875288; stNO_LENS[559].fHigh := 37.613499; 
    stNO_LENS[560].fEnergy := 15536.582147; stNO_LENS[560].fLow := 15.813813; stNO_LENS[560].fHigh := 37.466308; 
    stNO_LENS[561].fEnergy := 15567.686405; stNO_LENS[561].fLow := 15.752602; stNO_LENS[561].fHigh := 37.319631; 
    stNO_LENS[562].fEnergy := 15598.852934; stNO_LENS[562].fLow := 15.691652; stNO_LENS[562].fHigh := 37.173465; 
    stNO_LENS[563].fEnergy := 15630.081858; stNO_LENS[563].fLow := 15.630963; stNO_LENS[563].fHigh := 37.027810; 
    stNO_LENS[564].fEnergy := 15661.373303; stNO_LENS[564].fLow := 15.570534; stNO_LENS[564].fHigh := 36.882662; 
    stNO_LENS[565].fEnergy := 15692.727393; stNO_LENS[565].fLow := 15.510362; stNO_LENS[565].fHigh := 36.738020; 
    stNO_LENS[566].fEnergy := 15724.144254; stNO_LENS[566].fLow := 15.450448; stNO_LENS[566].fHigh := 36.593881; 
    stNO_LENS[567].fEnergy := 15755.624012; stNO_LENS[567].fLow := 15.390789; stNO_LENS[567].fHigh := 36.450243; 
    stNO_LENS[568].fEnergy := 15787.166792; stNO_LENS[568].fLow := 15.331386; stNO_LENS[568].fHigh := 36.307103; 
    stNO_LENS[569].fEnergy := 15818.772721; stNO_LENS[569].fLow := 15.272235; stNO_LENS[569].fHigh := 36.164461; 
    stNO_LENS[570].fEnergy := 15850.441925; stNO_LENS[570].fLow := 15.213337; stNO_LENS[570].fHigh := 36.022313; 
    stNO_LENS[571].fEnergy := 15882.174531; stNO_LENS[571].fLow := 15.154690; stNO_LENS[571].fHigh := 35.880657; 
    stNO_LENS[572].fEnergy := 15913.970666; stNO_LENS[572].fLow := 15.096292; stNO_LENS[572].fHigh := 35.739492; 
    stNO_LENS[573].fEnergy := 15945.830456; stNO_LENS[573].fLow := 15.038143; stNO_LENS[573].fHigh := 35.598816; 
    stNO_LENS[574].fEnergy := 15977.754030; stNO_LENS[574].fLow := 14.980242; stNO_LENS[574].fHigh := 35.458626; 
    stNO_LENS[575].fEnergy := 16009.741515; stNO_LENS[575].fLow := 14.922587; stNO_LENS[575].fHigh := 35.318921; 
    stNO_LENS[576].fEnergy := 16041.793039; stNO_LENS[576].fLow := 14.865177; stNO_LENS[576].fHigh := 35.179699; 
    stNO_LENS[577].fEnergy := 16073.908730; stNO_LENS[577].fLow := 14.808011; stNO_LENS[577].fHigh := 35.040958; 
    stNO_LENS[578].fEnergy := 16106.088717; stNO_LENS[578].fLow := 14.751088; stNO_LENS[578].fHigh := 34.902696; 
    stNO_LENS[579].fEnergy := 16138.333128; stNO_LENS[579].fLow := 14.694407; stNO_LENS[579].fHigh := 34.764912; 
    stNO_LENS[580].fEnergy := 16170.642092; stNO_LENS[580].fLow := 14.637966; stNO_LENS[580].fHigh := 34.627603; 
    stNO_LENS[581].fEnergy := 16203.015739; stNO_LENS[581].fLow := 14.581765; stNO_LENS[581].fHigh := 34.490768; 
    stNO_LENS[582].fEnergy := 16235.454198; stNO_LENS[582].fLow := 14.525802; stNO_LENS[582].fHigh := 34.354405; 
    stNO_LENS[583].fEnergy := 16267.957599; stNO_LENS[583].fLow := 14.470076; stNO_LENS[583].fHigh := 34.218513; 
    stNO_LENS[584].fEnergy := 16300.526072; stNO_LENS[584].fLow := 14.414586; stNO_LENS[584].fHigh := 34.083090; 
    stNO_LENS[585].fEnergy := 16333.159747; stNO_LENS[585].fLow := 14.359331; stNO_LENS[585].fHigh := 33.948135; 
    stNO_LENS[586].fEnergy := 16365.858755; stNO_LENS[586].fLow := 14.304310; stNO_LENS[586].fHigh := 33.813645; 
    stNO_LENS[587].fEnergy := 16398.623226; stNO_LENS[587].fLow := 14.249522; stNO_LENS[587].fHigh := 33.679620; 
    stNO_LENS[588].fEnergy := 16431.453291; stNO_LENS[588].fLow := 14.194965; stNO_LENS[588].fHigh := 33.546059; 
    stNO_LENS[589].fEnergy := 16464.349083; stNO_LENS[589].fLow := 14.140639; stNO_LENS[589].fHigh := 33.412958; 
    stNO_LENS[590].fEnergy := 16497.310732; stNO_LENS[590].fLow := 14.086542; stNO_LENS[590].fHigh := 33.280318; 
    stNO_LENS[591].fEnergy := 16530.338370; stNO_LENS[591].fLow := 14.032673; stNO_LENS[591].fHigh := 33.148137; 
    stNO_LENS[592].fEnergy := 16563.432129; stNO_LENS[592].fLow := 13.979032; stNO_LENS[592].fHigh := 33.016414; 
    stNO_LENS[593].fEnergy := 16596.592142; stNO_LENS[593].fLow := 13.925617; stNO_LENS[593].fHigh := 32.885146; 
    stNO_LENS[594].fEnergy := 16629.818542; stNO_LENS[594].fLow := 13.872427; stNO_LENS[594].fHigh := 32.754334; 
    stNO_LENS[595].fEnergy := 16663.111461; stNO_LENS[595].fLow := 13.819461; stNO_LENS[595].fHigh := 32.623976; 
    stNO_LENS[596].fEnergy := 16696.471032; stNO_LENS[596].fLow := 13.766718; stNO_LENS[596].fHigh := 32.494070; 
    stNO_LENS[597].fEnergy := 16729.897390; stNO_LENS[597].fLow := 13.714197; stNO_LENS[597].fHigh := 32.364616; 
    stNO_LENS[598].fEnergy := 16763.390666; stNO_LENS[598].fLow := 13.661897; stNO_LENS[598].fHigh := 32.235612; 
    stNO_LENS[599].fEnergy := 16796.950997; stNO_LENS[599].fLow := 13.609816; stNO_LENS[599].fHigh := 32.107058; 
    stNO_LENS[600].fEnergy := 16830.578515; stNO_LENS[600].fLow := 13.557955; stNO_LENS[600].fHigh := 31.978951; 
    stNO_LENS[601].fEnergy := 16864.273356; stNO_LENS[601].fLow := 13.506311; stNO_LENS[601].fHigh := 31.851292; 
    stNO_LENS[602].fEnergy := 16898.035654; stNO_LENS[602].fLow := 13.454884; stNO_LENS[602].fHigh := 31.724080; 
    stNO_LENS[603].fEnergy := 16931.865544; stNO_LENS[603].fLow := 13.403673; stNO_LENS[603].fHigh := 31.597312; 
    stNO_LENS[604].fEnergy := 16965.763161; stNO_LENS[604].fLow := 13.352676; stNO_LENS[604].fHigh := 31.470989; 
    stNO_LENS[605].fEnergy := 16999.728641; stNO_LENS[605].fLow := 13.301893; stNO_LENS[605].fHigh := 31.345109; 
    stNO_LENS[606].fEnergy := 17033.762121; stNO_LENS[606].fLow := 13.251323; stNO_LENS[606].fHigh := 31.219671; 
    stNO_LENS[607].fEnergy := 17067.863735; stNO_LENS[607].fLow := 13.200964; stNO_LENS[607].fHigh := 31.094676; 
    stNO_LENS[608].fEnergy := 17102.033621; stNO_LENS[608].fLow := 13.150816; stNO_LENS[608].fHigh := 30.970121; 
    stNO_LENS[609].fEnergy := 17136.271915; stNO_LENS[609].fLow := 13.100878; stNO_LENS[609].fHigh := 30.846006; 
    stNO_LENS[610].fEnergy := 17170.578755; stNO_LENS[610].fLow := 13.051148; stNO_LENS[610].fHigh := 30.722330; 
    stNO_LENS[611].fEnergy := 17204.954276; stNO_LENS[611].fLow := 13.001626; stNO_LENS[611].fHigh := 30.599092; 
    stNO_LENS[612].fEnergy := 17239.398618; stNO_LENS[612].fLow := 12.952310; stNO_LENS[612].fHigh := 30.476292; 
    stNO_LENS[613].fEnergy := 17273.911917; stNO_LENS[613].fLow := 12.903201; stNO_LENS[613].fHigh := 30.353929; 
    stNO_LENS[614].fEnergy := 17308.494311; stNO_LENS[614].fLow := 12.854296; stNO_LENS[614].fHigh := 30.232002; 
    stNO_LENS[615].fEnergy := 17343.145940; stNO_LENS[615].fLow := 12.805595; stNO_LENS[615].fHigh := 30.110511; 
    stNO_LENS[616].fEnergy := 17377.866941; stNO_LENS[616].fLow := 12.757096; stNO_LENS[616].fHigh := 29.989454; 
    stNO_LENS[617].fEnergy := 17412.657454; stNO_LENS[617].fLow := 12.708800; stNO_LENS[617].fHigh := 29.868832; 
    stNO_LENS[618].fEnergy := 17447.517618; stNO_LENS[618].fLow := 12.660704; stNO_LENS[618].fHigh := 29.748643; 
    stNO_LENS[619].fEnergy := 17482.447571; stNO_LENS[619].fLow := 12.612808; stNO_LENS[619].fHigh := 29.628886; 
    stNO_LENS[620].fEnergy := 17517.447455; stNO_LENS[620].fLow := 12.565111; stNO_LENS[620].fHigh := 29.509562; 
    stNO_LENS[621].fEnergy := 17552.517408; stNO_LENS[621].fLow := 12.517613; stNO_LENS[621].fHigh := 29.390670; 
    stNO_LENS[622].fEnergy := 17587.657571; stNO_LENS[622].fLow := 12.470311; stNO_LENS[622].fHigh := 29.272208; 
    stNO_LENS[623].fEnergy := 17622.868085; stNO_LENS[623].fLow := 12.423205; stNO_LENS[623].fHigh := 29.154177; 
    stNO_LENS[624].fEnergy := 17658.149090; stNO_LENS[624].fLow := 12.376295; stNO_LENS[624].fHigh := 29.036576; 
    stNO_LENS[625].fEnergy := 17693.500728; stNO_LENS[625].fLow := 12.329579; stNO_LENS[625].fHigh := 28.919403; 
    stNO_LENS[626].fEnergy := 17728.923140; stNO_LENS[626].fLow := 12.283057; stNO_LENS[626].fHigh := 28.802660; 
    stNO_LENS[627].fEnergy := 17764.416468; stNO_LENS[627].fLow := 12.236727; stNO_LENS[627].fHigh := 28.686344; 
    stNO_LENS[628].fEnergy := 17799.980854; stNO_LENS[628].fLow := 12.190588; stNO_LENS[628].fHigh := 28.570455; 
    stNO_LENS[629].fEnergy := 17835.616439; stNO_LENS[629].fLow := 12.144640; stNO_LENS[629].fHigh := 28.454994; 
    stNO_LENS[630].fEnergy := 17871.323367; stNO_LENS[630].fLow := 12.098882; stNO_LENS[630].fHigh := 28.339959; 
    stNO_LENS[631].fEnergy := 17907.101780; stNO_LENS[631].fLow := 12.053313; stNO_LENS[631].fHigh := 28.225350; 
    stNO_LENS[632].fEnergy := 17942.951822; stNO_LENS[632].fLow := 12.007932; stNO_LENS[632].fHigh := 28.111165; 
    stNO_LENS[633].fEnergy := 17978.873635; stNO_LENS[633].fLow := 11.962737; stNO_LENS[633].fHigh := 27.997406; 
    stNO_LENS[634].fEnergy := 18014.867364; stNO_LENS[634].fLow := 11.917729; stNO_LENS[634].fHigh := 27.884070; 
    stNO_LENS[635].fEnergy := 18050.933153; stNO_LENS[635].fLow := 11.872906; stNO_LENS[635].fHigh := 27.771158; 
    stNO_LENS[636].fEnergy := 18087.071145; stNO_LENS[636].fLow := 11.828268; stNO_LENS[636].fHigh := 27.658668; 
    stNO_LENS[637].fEnergy := 18123.281486; stNO_LENS[637].fLow := 11.783813; stNO_LENS[637].fHigh := 27.546601; 
    stNO_LENS[638].fEnergy := 18159.564319; stNO_LENS[638].fLow := 11.739541; stNO_LENS[638].fHigh := 27.434956; 
    stNO_LENS[639].fEnergy := 18195.919791; stNO_LENS[639].fLow := 11.695451; stNO_LENS[639].fHigh := 27.323731; 
    stNO_LENS[640].fEnergy := 18232.348047; stNO_LENS[640].fLow := 11.651542; stNO_LENS[640].fHigh := 27.212927; 
    stNO_LENS[641].fEnergy := 18268.849232; stNO_LENS[641].fLow := 11.607812; stNO_LENS[641].fHigh := 27.102543; 
    stNO_LENS[642].fEnergy := 18305.423493; stNO_LENS[642].fLow := 11.564262; stNO_LENS[642].fHigh := 26.992577; 
    stNO_LENS[643].fEnergy := 18342.070975; stNO_LENS[643].fLow := 11.520891; stNO_LENS[643].fHigh := 26.883030; 
    stNO_LENS[644].fEnergy := 18378.791826; stNO_LENS[644].fLow := 11.477697; stNO_LENS[644].fHigh := 26.773901; 
    stNO_LENS[645].fEnergy := 18415.586191; stNO_LENS[645].fLow := 11.434679; stNO_LENS[645].fHigh := 26.665189; 
    stNO_LENS[646].fEnergy := 18452.454219; stNO_LENS[646].fLow := 11.391838; stNO_LENS[646].fHigh := 26.556894; 
    stNO_LENS[647].fEnergy := 18489.396057; stNO_LENS[647].fLow := 11.349171; stNO_LENS[647].fHigh := 26.449014; 
    stNO_LENS[648].fEnergy := 18526.411853; stNO_LENS[648].fLow := 11.306679; stNO_LENS[648].fHigh := 26.341549; 
    stNO_LENS[649].fEnergy := 18563.501754; stNO_LENS[649].fLow := 11.264360; stNO_LENS[649].fHigh := 26.234498; 
    stNO_LENS[650].fEnergy := 18600.665909; stNO_LENS[650].fLow := 11.222214; stNO_LENS[650].fHigh := 26.127860; 
    stNO_LENS[651].fEnergy := 18637.904467; stNO_LENS[651].fLow := 11.180239; stNO_LENS[651].fHigh := 26.021634; 
    stNO_LENS[652].fEnergy := 18675.217577; stNO_LENS[652].fLow := 11.138436; stNO_LENS[652].fHigh := 25.915821; 
    stNO_LENS[653].fEnergy := 18712.605388; stNO_LENS[653].fLow := 11.096802; stNO_LENS[653].fHigh := 25.810418; 
    stNO_LENS[654].fEnergy := 18750.068048; stNO_LENS[654].fLow := 11.055338; stNO_LENS[654].fHigh := 25.705425; 
    stNO_LENS[655].fEnergy := 18787.605710; stNO_LENS[655].fLow := 11.014042; stNO_LENS[655].fHigh := 25.600840; 
    stNO_LENS[656].fEnergy := 18825.218521; stNO_LENS[656].fLow := 10.972914; stNO_LENS[656].fHigh := 25.496664; 
    stNO_LENS[657].fEnergy := 18862.906634; stNO_LENS[657].fLow := 10.931953; stNO_LENS[657].fHigh := 25.392895; 
    stNO_LENS[658].fEnergy := 18900.670198; stNO_LENS[658].fLow := 10.891158; stNO_LENS[658].fHigh := 25.289532; 
    stNO_LENS[659].fEnergy := 18938.509365; stNO_LENS[659].fLow := 10.850529; stNO_LENS[659].fHigh := 25.186573; 
    stNO_LENS[660].fEnergy := 18976.424286; stNO_LENS[660].fLow := 10.810064; stNO_LENS[660].fHigh := 25.084019; 
    stNO_LENS[661].fEnergy := 19014.415113; stNO_LENS[661].fLow := 10.769763; stNO_LENS[661].fHigh := 24.981867; 
    stNO_LENS[662].fEnergy := 19052.481997; stNO_LENS[662].fLow := 10.729624; stNO_LENS[662].fHigh := 24.880116; 
    stNO_LENS[663].fEnergy := 19090.625092; stNO_LENS[663].fLow := 10.689649; stNO_LENS[663].fHigh := 24.778766; 
    stNO_LENS[664].fEnergy := 19128.844549; stNO_LENS[664].fLow := 10.649834; stNO_LENS[664].fHigh := 24.677815; 
    stNO_LENS[665].fEnergy := 19167.140521; stNO_LENS[665].fLow := 10.610180; stNO_LENS[665].fHigh := 24.577262; 
    stNO_LENS[666].fEnergy := 19205.513162; stNO_LENS[666].fLow := 10.570686; stNO_LENS[666].fHigh := 24.477105; 
    stNO_LENS[667].fEnergy := 19243.962625; stNO_LENS[667].fLow := 10.531352; stNO_LENS[667].fHigh := 24.377344; 
    stNO_LENS[668].fEnergy := 19282.489064; stNO_LENS[668].fLow := 10.492176; stNO_LENS[668].fHigh := 24.277976; 
    stNO_LENS[669].fEnergy := 19321.092632; stNO_LENS[669].fLow := 10.453157; stNO_LENS[669].fHigh := 24.179000; 
    stNO_LENS[670].fEnergy := 19359.773486; stNO_LENS[670].fLow := 10.414296; stNO_LENS[670].fHigh := 24.080416; 
    stNO_LENS[671].fEnergy := 19398.531778; stNO_LENS[671].fLow := 10.375590; stNO_LENS[671].fHigh := 23.982220; 
    stNO_LENS[672].fEnergy := 19437.367665; stNO_LENS[672].fLow := 10.337040; stNO_LENS[672].fHigh := 23.884412; 
    stNO_LENS[673].fEnergy := 19476.281301; stNO_LENS[673].fLow := 10.298645; stNO_LENS[673].fHigh := 23.786991; 
    stNO_LENS[674].fEnergy := 19515.272842; stNO_LENS[674].fLow := 10.260404; stNO_LENS[674].fHigh := 23.689953; 
    stNO_LENS[675].fEnergy := 19554.342444; stNO_LENS[675].fLow := 10.222316; stNO_LENS[675].fHigh := 23.593298; 
    stNO_LENS[676].fEnergy := 19593.490264; stNO_LENS[676].fLow := 10.184381; stNO_LENS[676].fHigh := 23.497024; 
    stNO_LENS[677].fEnergy := 19632.716457; stNO_LENS[677].fLow := 10.146598; stNO_LENS[677].fHigh := 23.401130; 
    stNO_LENS[678].fEnergy := 19672.021182; stNO_LENS[678].fLow := 10.108965; stNO_LENS[678].fHigh := 23.305612; 
    stNO_LENS[679].fEnergy := 19711.404594; stNO_LENS[679].fLow := 10.071483; stNO_LENS[679].fHigh := 23.210469; 
    stNO_LENS[680].fEnergy := 19750.866853; stNO_LENS[680].fLow := 10.034151; stNO_LENS[680].fHigh := 23.115700; 
    stNO_LENS[681].fEnergy := 19790.408115; stNO_LENS[681].fLow := 9.996968; stNO_LENS[681].fHigh := 23.021302; 
    stNO_LENS[682].fEnergy := 19830.028538; stNO_LENS[682].fLow := 9.959933; stNO_LENS[682].fHigh := 22.927272; 
    stNO_LENS[683].fEnergy := 19869.728282; stNO_LENS[683].fLow := 9.923045; stNO_LENS[683].fHigh := 22.833610; 
    stNO_LENS[684].fEnergy := 19909.507504; stNO_LENS[684].fLow := 9.886305; stNO_LENS[684].fHigh := 22.740313; 
    stNO_LENS[685].fEnergy := 19949.366365; stNO_LENS[685].fLow := 9.849710; stNO_LENS[685].fHigh := 22.647377; 
    stNO_LENS[686].fEnergy := 19989.305023; stNO_LENS[686].fLow := 9.813261; stNO_LENS[686].fHigh := 22.554802; 
    stNO_LENS[687].fEnergy := 20029.323638; stNO_LENS[687].fLow := 9.776957; stNO_LENS[687].fHigh := 22.462584; 
    stNO_LENS[688].fEnergy := 20069.422371; stNO_LENS[688].fLow := 9.740797; stNO_LENS[688].fHigh := 22.370722; 
    stNO_LENS[689].fEnergy := 20109.601381; stNO_LENS[689].fLow := 9.704781; stNO_LENS[689].fHigh := 22.279212; 
    stNO_LENS[690].fEnergy := 20149.860830; stNO_LENS[690].fLow := 9.668907; stNO_LENS[690].fHigh := 22.188052; 
    stNO_LENS[691].fEnergy := 20190.200878; stNO_LENS[691].fLow := 9.633176; stNO_LENS[691].fHigh := 22.097240; 
    stNO_LENS[692].fEnergy := 20230.621687; stNO_LENS[692].fLow := 9.597585; stNO_LENS[692].fHigh := 22.006772; 
    stNO_LENS[693].fEnergy := 20271.123419; stNO_LENS[693].fLow := 9.562136; stNO_LENS[693].fHigh := 21.916647; 
    stNO_LENS[694].fEnergy := 20311.706235; stNO_LENS[694].fLow := 9.526827; stNO_LENS[694].fHigh := 21.826860; 
    stNO_LENS[695].fEnergy := 20352.370298; stNO_LENS[695].fLow := 9.491657; stNO_LENS[695].fHigh := 21.737409; 
    stNO_LENS[696].fEnergy := 20393.115770; stNO_LENS[696].fLow := 9.456626; stNO_LENS[696].fHigh := 21.648292; 
    stNO_LENS[697].fEnergy := 20433.942815; stNO_LENS[697].fLow := 9.421733; stNO_LENS[697].fHigh := 21.559504; 
    stNO_LENS[698].fEnergy := 20474.851596; stNO_LENS[698].fLow := 9.386977; stNO_LENS[698].fHigh := 21.471043; 
    stNO_LENS[699].fEnergy := 20515.842276; stNO_LENS[699].fLow := 9.352359; stNO_LENS[699].fHigh := 21.382907; 
    stNO_LENS[700].fEnergy := 20556.915020; stNO_LENS[700].fLow := 9.317876; stNO_LENS[700].fHigh := 21.295090; 
    stNO_LENS[701].fEnergy := 20598.069991; stNO_LENS[701].fLow := 9.283529; stNO_LENS[701].fHigh := 21.207591; 
    stNO_LENS[702].fEnergy := 20639.307355; stNO_LENS[702].fLow := 9.249317; stNO_LENS[702].fHigh := 21.120406; 
    stNO_LENS[703].fEnergy := 20680.627276; stNO_LENS[703].fLow := 9.215240; stNO_LENS[703].fHigh := 21.033530; 
    stNO_LENS[704].fEnergy := 20722.029919; stNO_LENS[704].fLow := 9.181296; stNO_LENS[704].fHigh := 20.946962; 
    stNO_LENS[705].fEnergy := 20763.515451; stNO_LENS[705].fLow := 9.147485; stNO_LENS[705].fHigh := 20.860696; 
    stNO_LENS[706].fEnergy := 20805.084036; stNO_LENS[706].fLow := 9.113806; stNO_LENS[706].fHigh := 20.774730; 
    stNO_LENS[707].fEnergy := 20846.735842; stNO_LENS[707].fLow := 9.080259; stNO_LENS[707].fHigh := 20.689059; 
    stNO_LENS[708].fEnergy := 20888.471035; stNO_LENS[708].fLow := 9.046843; stNO_LENS[708].fHigh := 20.603681; 
    stNO_LENS[709].fEnergy := 20930.289782; stNO_LENS[709].fLow := 9.013558; stNO_LENS[709].fHigh := 20.518590; 
    stNO_LENS[710].fEnergy := 20972.192250; stNO_LENS[710].fLow := 8.980403; stNO_LENS[710].fHigh := 20.433782; 
    stNO_LENS[711].fEnergy := 21014.178607; stNO_LENS[711].fLow := 8.947377; stNO_LENS[711].fHigh := 20.349255; 
    stNO_LENS[712].fEnergy := 21056.249021; stNO_LENS[712].fLow := 8.914480; stNO_LENS[712].fHigh := 20.265003; 
    stNO_LENS[713].fEnergy := 21098.403659; stNO_LENS[713].fLow := 8.881710; stNO_LENS[713].fHigh := 20.181022; 
    stNO_LENS[714].fEnergy := 21140.642692; stNO_LENS[714].fLow := 8.849069; stNO_LENS[714].fHigh := 20.097308; 
    stNO_LENS[715].fEnergy := 21182.966286; stNO_LENS[715].fLow := 8.816554; stNO_LENS[715].fHigh := 20.013857; 
    stNO_LENS[716].fEnergy := 21225.374613; stNO_LENS[716].fLow := 8.784166; stNO_LENS[716].fHigh := 19.930664; 
    stNO_LENS[717].fEnergy := 21267.867841; stNO_LENS[717].fLow := 8.751903; stNO_LENS[717].fHigh := 19.847725; 
    stNO_LENS[718].fEnergy := 21310.446141; stNO_LENS[718].fLow := 8.719765; stNO_LENS[718].fHigh := 19.765034; 
    stNO_LENS[719].fEnergy := 21353.109683; stNO_LENS[719].fLow := 8.687752; stNO_LENS[719].fHigh := 19.682588; 
    stNO_LENS[720].fEnergy := 21395.858637; stNO_LENS[720].fLow := 8.655863; stNO_LENS[720].fHigh := 19.600381; 
    stNO_LENS[721].fEnergy := 21438.693174; stNO_LENS[721].fLow := 8.624097; stNO_LENS[721].fHigh := 19.518409; 
    stNO_LENS[722].fEnergy := 21481.613467; stNO_LENS[722].fLow := 8.592454; stNO_LENS[722].fHigh := 19.436667; 
    stNO_LENS[723].fEnergy := 21524.619686; stNO_LENS[723].fLow := 8.560934; stNO_LENS[723].fHigh := 19.355149; 
    stNO_LENS[724].fEnergy := 21567.712003; stNO_LENS[724].fLow := 8.529535; stNO_LENS[724].fHigh := 19.273850; 
    stNO_LENS[725].fEnergy := 21610.890591; stNO_LENS[725].fLow := 8.498257; stNO_LENS[725].fHigh := 19.192766; 
    stNO_LENS[726].fEnergy := 21654.155623; stNO_LENS[726].fLow := 8.467099; stNO_LENS[726].fHigh := 19.111891; 
    stNO_LENS[727].fEnergy := 21697.507271; stNO_LENS[727].fLow := 8.436062; stNO_LENS[727].fHigh := 19.031220; 
    stNO_LENS[728].fEnergy := 21740.945710; stNO_LENS[728].fLow := 8.405143; stNO_LENS[728].fHigh := 18.950747; 
    stNO_LENS[729].fEnergy := 21784.471112; stNO_LENS[729].fLow := 8.374344; stNO_LENS[729].fHigh := 18.870467; 
    stNO_LENS[730].fEnergy := 21828.083652; stNO_LENS[730].fLow := 8.343663; stNO_LENS[730].fHigh := 18.790374; 
    stNO_LENS[731].fEnergy := 21871.783505; stNO_LENS[731].fLow := 8.313100; stNO_LENS[731].fHigh := 18.710462; 
    stNO_LENS[732].fEnergy := 21915.570845; stNO_LENS[732].fLow := 8.282654; stNO_LENS[732].fHigh := 18.630727; 
    stNO_LENS[733].fEnergy := 21959.445847; stNO_LENS[733].fLow := 8.252324; stNO_LENS[733].fHigh := 18.551161; 
    stNO_LENS[734].fEnergy := 22003.408687; stNO_LENS[734].fLow := 8.222111; stNO_LENS[734].fHigh := 18.471760; 
    stNO_LENS[735].fEnergy := 22047.459540; stNO_LENS[735].fLow := 8.192013; stNO_LENS[735].fHigh := 18.392516; 
    stNO_LENS[736].fEnergy := 22091.598584; stNO_LENS[736].fLow := 8.162030; stNO_LENS[736].fHigh := 18.313425; 
    stNO_LENS[737].fEnergy := 22135.825994; stNO_LENS[737].fLow := 8.132161; stNO_LENS[737].fHigh := 18.234480; 
    stNO_LENS[738].fEnergy := 22180.141947; stNO_LENS[738].fLow := 8.102407; stNO_LENS[738].fHigh := 18.155674; 
    stNO_LENS[739].fEnergy := 22224.546620; stNO_LENS[739].fLow := 8.072766; stNO_LENS[739].fHigh := 18.077002; 
    stNO_LENS[740].fEnergy := 22269.040192; stNO_LENS[740].fLow := 8.043238; stNO_LENS[740].fHigh := 17.998456; 
    stNO_LENS[741].fEnergy := 22313.622841; stNO_LENS[741].fLow := 8.013822; stNO_LENS[741].fHigh := 17.920032; 
    stNO_LENS[742].fEnergy := 22358.294743; stNO_LENS[742].fLow := 7.984518; stNO_LENS[742].fHigh := 17.841721; 
    stNO_LENS[743].fEnergy := 22403.056079; stNO_LENS[743].fLow := 7.955325; stNO_LENS[743].fHigh := 17.763519; 
    stNO_LENS[744].fEnergy := 22447.907027; stNO_LENS[744].fLow := 7.926243; stNO_LENS[744].fHigh := 17.685417; 
    stNO_LENS[745].fEnergy := 22492.847767; stNO_LENS[745].fLow := 7.897271; stNO_LENS[745].fHigh := 17.607409; 
    stNO_LENS[746].fEnergy := 22537.878478; stNO_LENS[746].fLow := 7.868409; stNO_LENS[746].fHigh := 17.529489; 
    stNO_LENS[747].fEnergy := 22582.999341; stNO_LENS[747].fLow := 7.839657; stNO_LENS[747].fHigh := 17.451649; 
    stNO_LENS[748].fEnergy := 22628.210536; stNO_LENS[748].fLow := 7.811013; stNO_LENS[748].fHigh := 17.373883; 
    stNO_LENS[749].fEnergy := 22673.512244; stNO_LENS[749].fLow := 7.782477; stNO_LENS[749].fHigh := 17.296183; 
    stNO_LENS[750].fEnergy := 22718.904645; stNO_LENS[750].fLow := 7.754049; stNO_LENS[750].fHigh := 17.218543; 
    stNO_LENS[751].fEnergy := 22764.387923; stNO_LENS[751].fLow := 7.725728; stNO_LENS[751].fHigh := 17.140955; 
    stNO_LENS[752].fEnergy := 22809.962258; stNO_LENS[752].fLow := 7.697514; stNO_LENS[752].fHigh := 17.063413; 
    stNO_LENS[753].fEnergy := 22855.627833; stNO_LENS[753].fLow := 7.669406; stNO_LENS[753].fHigh := 16.985908; 
    stNO_LENS[754].fEnergy := 22901.384830; stNO_LENS[754].fLow := 7.641404; stNO_LENS[754].fHigh := 16.908434; 
    stNO_LENS[755].fEnergy := 22947.233433; stNO_LENS[755].fLow := 7.613508; stNO_LENS[755].fHigh := 16.830984; 
    stNO_LENS[756].fEnergy := 22993.173825; stNO_LENS[756].fLow := 7.585716; stNO_LENS[756].fHigh := 16.753549; 
    stNO_LENS[757].fEnergy := 23039.206190; stNO_LENS[757].fLow := 7.558028; stNO_LENS[757].fHigh := 16.676123; 
    stNO_LENS[758].fEnergy := 23085.330711; stNO_LENS[758].fLow := 7.530444; stNO_LENS[758].fHigh := 16.598698; 
    stNO_LENS[759].fEnergy := 23131.547574; stNO_LENS[759].fLow := 7.502963; stNO_LENS[759].fHigh := 16.521266; 
    stNO_LENS[760].fEnergy := 23177.856963; stNO_LENS[760].fLow := 7.475586; stNO_LENS[760].fHigh := 16.443819; 
    stNO_LENS[761].fEnergy := 23224.259064; stNO_LENS[761].fLow := 7.448310; stNO_LENS[761].fHigh := 16.366351; 
    stNO_LENS[762].fEnergy := 23270.754061; stNO_LENS[762].fLow := 7.421137; stNO_LENS[762].fHigh := 16.288853; 
    stNO_LENS[763].fEnergy := 23317.342142; stNO_LENS[763].fLow := 7.394065; stNO_LENS[763].fHigh := 16.211317; 
    stNO_LENS[764].fEnergy := 23364.023492; stNO_LENS[764].fLow := 7.367093; stNO_LENS[764].fHigh := 16.133736; 
    stNO_LENS[765].fEnergy := 23410.798298; stNO_LENS[765].fLow := 7.340223; stNO_LENS[765].fHigh := 16.056102; 
    stNO_LENS[766].fEnergy := 23457.666748; stNO_LENS[766].fLow := 7.313452; stNO_LENS[766].fHigh := 15.931383; 
    stNO_LENS[767].fEnergy := 23504.629028; stNO_LENS[767].fLow := 7.286781; stNO_LENS[767].fHigh := 15.863347; 
    stNO_LENS[768].fEnergy := 23551.685327; stNO_LENS[768].fLow := 7.260209; stNO_LENS[768].fHigh := 15.795576; 
    stNO_LENS[769].fEnergy := 23598.835832; stNO_LENS[769].fLow := 7.233736; stNO_LENS[769].fHigh := 15.728069; 
    stNO_LENS[770].fEnergy := 23646.080733; stNO_LENS[770].fLow := 7.207361; stNO_LENS[770].fHigh := 15.660825; 
    stNO_LENS[771].fEnergy := 23693.420218; stNO_LENS[771].fLow := 7.181083; stNO_LENS[771].fHigh := 15.593845; 
    stNO_LENS[772].fEnergy := 23740.854477; stNO_LENS[772].fLow := 7.154903; stNO_LENS[772].fHigh := 15.527128; 
    stNO_LENS[773].fEnergy := 23788.383699; stNO_LENS[773].fLow := 7.128820; stNO_LENS[773].fHigh := 15.460674; 
    stNO_LENS[774].fEnergy := 23836.008075; stNO_LENS[774].fLow := 7.102833; stNO_LENS[774].fHigh := 15.394481; 
    stNO_LENS[775].fEnergy := 23883.727795; stNO_LENS[775].fLow := 7.076942; stNO_LENS[775].fHigh := 15.328551; 
    stNO_LENS[776].fEnergy := 23931.543050; stNO_LENS[776].fLow := 7.051147; stNO_LENS[776].fHigh := 15.262881; 
    stNO_LENS[777].fEnergy := 23979.454031; stNO_LENS[777].fLow := 7.025446; stNO_LENS[777].fHigh := 15.197473; 
    stNO_LENS[778].fEnergy := 24027.460930; stNO_LENS[778].fLow := 6.999841; stNO_LENS[778].fHigh := 15.132325; 
    stNO_LENS[779].fEnergy := 24075.563939; stNO_LENS[779].fLow := 6.974329; stNO_LENS[779].fHigh := 15.067437; 
    stNO_LENS[780].fEnergy := 24123.763250; stNO_LENS[780].fLow := 6.948912; stNO_LENS[780].fHigh := 15.002808; 
    stNO_LENS[781].fEnergy := 24172.059056; stNO_LENS[781].fLow := 6.923587; stNO_LENS[781].fHigh := 14.938438; 
    stNO_LENS[782].fEnergy := 24220.451551; stNO_LENS[782].fLow := 6.898356; stNO_LENS[782].fHigh := 14.874327; 
    stNO_LENS[783].fEnergy := 24268.940927; stNO_LENS[783].fLow := 6.873217; stNO_LENS[783].fHigh := 14.810474; 
    stNO_LENS[784].fEnergy := 24317.527379; stNO_LENS[784].fLow := 6.848170; stNO_LENS[784].fHigh := 14.746878; 
    stNO_LENS[785].fEnergy := 24366.211101; stNO_LENS[785].fLow := 6.823215; stNO_LENS[785].fHigh := 14.683540; 
    stNO_LENS[786].fEnergy := 24414.992288; stNO_LENS[786].fLow := 6.798351; stNO_LENS[786].fHigh := 14.620458; 
    stNO_LENS[787].fEnergy := 24463.871136; stNO_LENS[787].fLow := 6.773577; stNO_LENS[787].fHigh := 14.557632; 
    stNO_LENS[788].fEnergy := 24512.847838; stNO_LENS[788].fLow := 6.748895; stNO_LENS[788].fHigh := 14.495062; 
    stNO_LENS[789].fEnergy := 24561.922592; stNO_LENS[789].fLow := 6.724302; stNO_LENS[789].fHigh := 14.432747; 
    stNO_LENS[790].fEnergy := 24611.095594; stNO_LENS[790].fLow := 6.699798; stNO_LENS[790].fHigh := 14.370686; 
    stNO_LENS[791].fEnergy := 24660.367040; stNO_LENS[791].fLow := 6.675384; stNO_LENS[791].fHigh := 14.308880; 
    stNO_LENS[792].fEnergy := 24709.737128; stNO_LENS[792].fLow := 6.651059; stNO_LENS[792].fHigh := 14.247327; 
    stNO_LENS[793].fEnergy := 24759.206055; stNO_LENS[793].fLow := 6.626822; stNO_LENS[793].fHigh := 14.186027; 
    stNO_LENS[794].fEnergy := 24808.774018; stNO_LENS[794].fLow := 6.602673; stNO_LENS[794].fHigh := 14.124980; 
    stNO_LENS[795].fEnergy := 24858.441217; stNO_LENS[795].fLow := 6.578611; stNO_LENS[795].fHigh := 14.064184; 
    stNO_LENS[796].fEnergy := 24908.207849; stNO_LENS[796].fLow := 6.554637; stNO_LENS[796].fHigh := 14.003640; 
    stNO_LENS[797].fEnergy := 24958.074115; stNO_LENS[797].fLow := 6.530749; stNO_LENS[797].fHigh := 13.943347; 
    stNO_LENS[798].fEnergy := 25008.040212; stNO_LENS[798].fLow := 6.506948; stNO_LENS[798].fHigh := 13.883304; 
    stNO_LENS[799].fEnergy := 25058.106342; stNO_LENS[799].fLow := 6.483233; stNO_LENS[799].fHigh := 13.823511; 
    stNO_LENS[800].fEnergy := 25108.272705; stNO_LENS[800].fLow := 6.459603; stNO_LENS[800].fHigh := 13.763967; 
    stNO_LENS[801].fEnergy := 25158.539500; stNO_LENS[801].fLow := 6.436058; stNO_LENS[801].fHigh := 13.704672; 
    stNO_LENS[802].fEnergy := 25208.906930; stNO_LENS[802].fLow := 6.412599; stNO_LENS[802].fHigh := 13.645625; 
    stNO_LENS[803].fEnergy := 25259.375195; stNO_LENS[803].fLow := 6.389223; stNO_LENS[803].fHigh := 13.586826; 
    stNO_LENS[804].fEnergy := 25309.944498; stNO_LENS[804].fLow := 6.365932; stNO_LENS[804].fHigh := 13.528273; 
    stNO_LENS[805].fEnergy := 25360.615041; stNO_LENS[805].fLow := 6.342724; stNO_LENS[805].fHigh := 13.469967; 
    stNO_LENS[806].fEnergy := 25411.387026; stNO_LENS[806].fLow := 6.319600; stNO_LENS[806].fHigh := 13.411907; 
    stNO_LENS[807].fEnergy := 25462.260656; stNO_LENS[807].fLow := 6.296559; stNO_LENS[807].fHigh := 13.354092; 
    stNO_LENS[808].fEnergy := 25513.236136; stNO_LENS[808].fLow := 6.273600; stNO_LENS[808].fHigh := 13.296522; 
    stNO_LENS[809].fEnergy := 25564.313669; stNO_LENS[809].fLow := 6.250723; stNO_LENS[809].fHigh := 13.239196; 
    stNO_LENS[810].fEnergy := 25615.493459; stNO_LENS[810].fLow := 6.227928; stNO_LENS[810].fHigh := 13.182113; 
    stNO_LENS[811].fEnergy := 25666.775711; stNO_LENS[811].fLow := 6.205214; stNO_LENS[811].fHigh := 13.125273; 
    stNO_LENS[812].fEnergy := 25718.160630; stNO_LENS[812].fLow := 6.182582; stNO_LENS[812].fHigh := 13.068676; 
    stNO_LENS[813].fEnergy := 25769.648422; stNO_LENS[813].fLow := 6.160030; stNO_LENS[813].fHigh := 13.012320; 
    stNO_LENS[814].fEnergy := 25821.239293; stNO_LENS[814].fLow := 6.137558; stNO_LENS[814].fHigh := 12.956206; 
    stNO_LENS[815].fEnergy := 25872.933448; stNO_LENS[815].fLow := 6.115167; stNO_LENS[815].fHigh := 12.900332; 
    stNO_LENS[816].fEnergy := 25924.731096; stNO_LENS[816].fLow := 6.092855; stNO_LENS[816].fHigh := 12.844697; 
    stNO_LENS[817].fEnergy := 25976.632442; stNO_LENS[817].fLow := 6.070622; stNO_LENS[817].fHigh := 12.789302; 
    stNO_LENS[818].fEnergy := 26028.637695; stNO_LENS[818].fLow := 6.048468; stNO_LENS[818].fHigh := 12.734146; 
    stNO_LENS[819].fEnergy := 26080.747062; stNO_LENS[819].fLow := 6.026393; stNO_LENS[819].fHigh := 12.679228; 
    stNO_LENS[820].fEnergy := 26132.960752; stNO_LENS[820].fLow := 6.004396; stNO_LENS[820].fHigh := 12.624547; 
    stNO_LENS[821].fEnergy := 26185.278975; stNO_LENS[821].fLow := 5.982477; stNO_LENS[821].fHigh := 12.570104; 
    stNO_LENS[822].fEnergy := 26237.701938; stNO_LENS[822].fLow := 5.960635; stNO_LENS[822].fHigh := 12.515896; 
    stNO_LENS[823].fEnergy := 26290.229852; stNO_LENS[823].fLow := 5.938870; stNO_LENS[823].fHigh := 12.461924; 
    stNO_LENS[824].fEnergy := 26342.862928; stNO_LENS[824].fLow := 5.917182; stNO_LENS[824].fHigh := 12.408187; 
    stNO_LENS[825].fEnergy := 26395.601374; stNO_LENS[825].fLow := 5.895571; stNO_LENS[825].fHigh := 12.354684; 
    stNO_LENS[826].fEnergy := 26448.445404; stNO_LENS[826].fLow := 5.874035; stNO_LENS[826].fHigh := 12.301415; 
    stNO_LENS[827].fEnergy := 26501.395226; stNO_LENS[827].fLow := 5.852576; stNO_LENS[827].fHigh := 12.248379; 
    stNO_LENS[828].fEnergy := 26554.451055; stNO_LENS[828].fLow := 5.831191; stNO_LENS[828].fHigh := 12.195575; 
    stNO_LENS[829].fEnergy := 26607.613102; stNO_LENS[829].fLow := 5.809882; stNO_LENS[829].fHigh := 12.143003; 
    stNO_LENS[830].fEnergy := 26660.881578; stNO_LENS[830].fLow := 5.788648; stNO_LENS[830].fHigh := 12.090662; 
    stNO_LENS[831].fEnergy := 26714.256699; stNO_LENS[831].fLow := 5.767488; stNO_LENS[831].fHigh := 12.038552; 
    stNO_LENS[832].fEnergy := 26767.738676; stNO_LENS[832].fLow := 5.746402; stNO_LENS[832].fHigh := 11.986672; 
    stNO_LENS[833].fEnergy := 26821.327725; stNO_LENS[833].fLow := 5.725390; stNO_LENS[833].fHigh := 11.935020; 
    stNO_LENS[834].fEnergy := 26875.024059; stNO_LENS[834].fLow := 5.704452; stNO_LENS[834].fHigh := 11.883598; 
    stNO_LENS[835].fEnergy := 26928.827893; stNO_LENS[835].fLow := 5.683586; stNO_LENS[835].fHigh := 11.832403; 
    stNO_LENS[836].fEnergy := 26982.739442; stNO_LENS[836].fLow := 5.662793; stNO_LENS[836].fHigh := 11.781435; 
    stNO_LENS[837].fEnergy := 27036.758923; stNO_LENS[837].fLow := 5.642073; stNO_LENS[837].fHigh := 11.730694; 
    stNO_LENS[838].fEnergy := 27090.886550; stNO_LENS[838].fLow := 5.621425; stNO_LENS[838].fHigh := 11.680179; 
    stNO_LENS[839].fEnergy := 27145.122541; stNO_LENS[839].fLow := 5.600849; stNO_LENS[839].fHigh := 11.629890; 
    stNO_LENS[840].fEnergy := 27199.467113; stNO_LENS[840].fLow := 5.580344; stNO_LENS[840].fHigh := 11.579824; 
    stNO_LENS[841].fEnergy := 27253.920482; stNO_LENS[841].fLow := 5.559911; stNO_LENS[841].fHigh := 11.529983; 
    stNO_LENS[842].fEnergy := 27308.482867; stNO_LENS[842].fLow := 5.539548; stNO_LENS[842].fHigh := 11.480365; 
    stNO_LENS[843].fEnergy := 27363.154486; stNO_LENS[843].fLow := 5.519256; stNO_LENS[843].fHigh := 11.430970; 
    stNO_LENS[844].fEnergy := 27417.935558; stNO_LENS[844].fLow := 5.499034; stNO_LENS[844].fHigh := 11.381797; 
    stNO_LENS[845].fEnergy := 27472.826302; stNO_LENS[845].fLow := 5.478882; stNO_LENS[845].fHigh := 11.332844; 
    stNO_LENS[846].fEnergy := 27527.826937; stNO_LENS[846].fLow := 5.458800; stNO_LENS[846].fHigh := 11.284113; 
    stNO_LENS[847].fEnergy := 27582.937683; stNO_LENS[847].fLow := 5.438787; stNO_LENS[847].fHigh := 11.235601; 
    stNO_LENS[848].fEnergy := 27638.158761; stNO_LENS[848].fLow := 5.418843; stNO_LENS[848].fHigh := 11.187309; 
    stNO_LENS[849].fEnergy := 27693.490392; stNO_LENS[849].fLow := 5.398968; stNO_LENS[849].fHigh := 11.139235; 
    stNO_LENS[850].fEnergy := 27748.932796; stNO_LENS[850].fLow := 5.379161; stNO_LENS[850].fHigh := 11.091380; 
    stNO_LENS[851].fEnergy := 27804.486197; stNO_LENS[851].fLow := 5.359422; stNO_LENS[851].fHigh := 11.043741; 
    stNO_LENS[852].fEnergy := 27860.150815; stNO_LENS[852].fLow := 5.339751; stNO_LENS[852].fHigh := 10.996319; 
    stNO_LENS[853].fEnergy := 27915.926874; stNO_LENS[853].fLow := 5.320148; stNO_LENS[853].fHigh := 10.949113; 
    stNO_LENS[854].fEnergy := 27971.814597; stNO_LENS[854].fLow := 5.300612; stNO_LENS[854].fHigh := 10.902122; 
    stNO_LENS[855].fEnergy := 28027.814207; stNO_LENS[855].fLow := 5.281143; stNO_LENS[855].fHigh := 10.855346; 
    stNO_LENS[856].fEnergy := 28083.925929; stNO_LENS[856].fLow := 5.261741; stNO_LENS[856].fHigh := 10.808784; 
    stNO_LENS[857].fEnergy := 28140.149986; stNO_LENS[857].fLow := 5.242405; stNO_LENS[857].fHigh := 10.762434; 
    stNO_LENS[858].fEnergy := 28196.486604; stNO_LENS[858].fLow := 5.223135; stNO_LENS[858].fHigh := 10.716298; 
    stNO_LENS[859].fEnergy := 28252.936008; stNO_LENS[859].fLow := 5.203930; stNO_LENS[859].fHigh := 10.670373; 
    stNO_LENS[860].fEnergy := 28309.498423; stNO_LENS[860].fLow := 5.184792; stNO_LENS[860].fHigh := 10.624659; 
    stNO_LENS[861].fEnergy := 28366.174077; stNO_LENS[861].fLow := 5.165718; stNO_LENS[861].fHigh := 10.579156; 
    stNO_LENS[862].fEnergy := 28422.963195; stNO_LENS[862].fLow := 5.146710; stNO_LENS[862].fHigh := 10.533862; 
    stNO_LENS[863].fEnergy := 28479.866005; stNO_LENS[863].fLow := 5.127766; stNO_LENS[863].fHigh := 10.488777; 
    stNO_LENS[864].fEnergy := 28536.882735; stNO_LENS[864].fLow := 5.108886; stNO_LENS[864].fHigh := 10.443901; 
    stNO_LENS[865].fEnergy := 28594.013612; stNO_LENS[865].fLow := 5.090071; stNO_LENS[865].fHigh := 10.399233; 
    stNO_LENS[866].fEnergy := 28651.258866; stNO_LENS[866].fLow := 5.071319; stNO_LENS[866].fHigh := 10.354771; 
    stNO_LENS[867].fEnergy := 28708.618724; stNO_LENS[867].fLow := 5.052631; stNO_LENS[867].fHigh := 10.310516; 
    stNO_LENS[868].fEnergy := 28766.093417; stNO_LENS[868].fLow := 5.034006; stNO_LENS[868].fHigh := 10.266467; 
    stNO_LENS[869].fEnergy := 28823.683175; stNO_LENS[869].fLow := 5.015445; stNO_LENS[869].fHigh := 10.222623; 
    stNO_LENS[870].fEnergy := 28881.388227; stNO_LENS[870].fLow := 4.996946; stNO_LENS[870].fHigh := 10.178982; 
    stNO_LENS[871].fEnergy := 28939.208804; stNO_LENS[871].fLow := 4.978509; stNO_LENS[871].fHigh := 10.135546; 
    stNO_LENS[872].fEnergy := 28997.145139; stNO_LENS[872].fLow := 4.960135; stNO_LENS[872].fHigh := 10.092312; 
    stNO_LENS[873].fEnergy := 29055.197462; stNO_LENS[873].fLow := 4.941822; stNO_LENS[873].fHigh := 10.049280; 
    stNO_LENS[874].fEnergy := 29113.366006; stNO_LENS[874].fLow := 4.923571; stNO_LENS[874].fHigh := 10.006450; 
    stNO_LENS[875].fEnergy := 29171.651004; stNO_LENS[875].fLow := 4.905382; stNO_LENS[875].fHigh := 9.963821; 
    stNO_LENS[876].fEnergy := 29230.052688; stNO_LENS[876].fLow := 4.887254; stNO_LENS[876].fHigh := 9.921392; 
    stNO_LENS[877].fEnergy := 29288.571293; stNO_LENS[877].fLow := 4.869186; stNO_LENS[877].fHigh := 9.879163; 
    stNO_LENS[878].fEnergy := 29347.207052; stNO_LENS[878].fLow := 4.851179; stNO_LENS[878].fHigh := 9.837132; 
    stNO_LENS[879].fEnergy := 29405.960199; stNO_LENS[879].fLow := 4.833233; stNO_LENS[879].fHigh := 9.795299; 
    stNO_LENS[880].fEnergy := 29464.830971; stNO_LENS[880].fLow := 4.815347; stNO_LENS[880].fHigh := 9.753664; 
